ABB RAPID module: Module1.mod

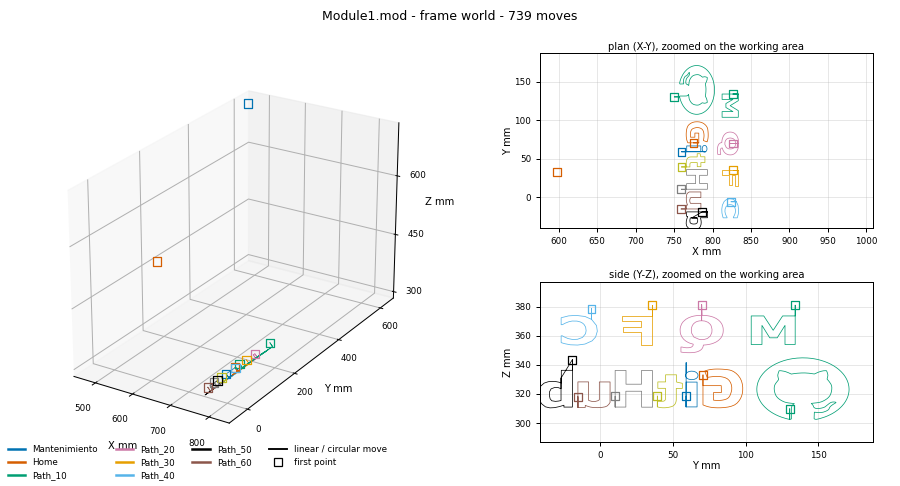
[picture p0: tool path of Module1.mod in frame world, 739 of 739 moves have a stored position in this frame; points joined in program order, loops and branches not executed]
MODULE Module1
    PERS tooldata TCP_Marcador:=[TRUE,[[70.711,0,142.836],[0.923879533,0,0.382683432,0]],[0.1,[0,0,1],[1,0,0,0],0,0,0]];
    PERS wobjdata Workobject_3:=[FALSE,TRUE,"",[[882.206,-55.622,379.617],[0.36650116,0,0.930417594,0]],[[0,0,0],[1,0,0,0]]];
    CONST robtarget Target_0:=[[81.772404685,689.476808944,-532.94398519],[0.776752007,-0.374117142,-0.504537271,-0.046204186],[0,0,-1,1],[9E+09,9E+09,9E+09,9E+09,9E+09,9E+09]];
    CONST robtarget Target_1:=[[84.162870332,88.825944226,-327.093570394],[0.96912891,0.008310335,0.246321364,-0.006773393],[0,-1,-1,0],[9E+09,9E+09,9E+09,9E+09,9E+09,9E+09]];
    CONST robtarget Target_50:=[[39.719,189.61,-28.8],[1,0,0,0],[-1,0,0,1],[9E+09,9E+09,9E+09,9E+09,9E+09,9E+09]];
    CONST robtarget Target_60:=[[39.719,180.982,-28.8],[1,0,0,0],[-1,0,0,1],[9E+09,9E+09,9E+09,9E+09,9E+09,9E+09]];
    CONST robtarget Target_70:=[[54.178,174.493,-28.8],[1,0,0,0],[-1,0,0,1],[9E+09,9E+09,9E+09,9E+09,9E+09,9E+09]];
    CONST robtarget Target_80:=[[39.719,168.028,-28.8],[1,0,0,0],[-1,0,0,1],[9E+09,9E+09,9E+09,9E+09,9E+09,9E+09]];
    CONST robtarget Target_180:=[[39.719,189.61,-38.8],[1,0,0,0],[-1,0,0,1],[9E+09,9E+09,9E+09,9E+09,9E+09,9E+09]];
    CONST robtarget Target_90:=[[39.719,159.4,-28.8],[1,0,0,0],[-1,0,0,1],[9E+09,9E+09,9E+09,9E+09,9E+09,9E+09]];
    CONST robtarget Target_100:=[[68.519,159.4,-28.8],[1,0,0,0],[-1,0,0,1],[9E+09,9E+09,9E+09,9E+09,9E+09,9E+09]];
    CONST robtarget Target_110:=[[68.519,166.782,-28.8],[1,0,0,0],[-1,0,0,1],[9E+09,9E+09,9E+09,9E+09,9E+09,9E+09]];
    CONST robtarget Target_120:=[[49.241,166.782,-28.8],[1,0,0,0],[-1,0,0,1],[9E+09,9E+09,9E+09,9E+09,9E+09,9E+09]];
    CONST robtarget Target_130:=[[61.748,172.119,-28.8],[1,0,0,0],[-1,0,0,1],[9E+09,9E+09,9E+09,9E+09,9E+09,9E+09]];
    CONST robtarget Target_140:=[[61.748,177.267,-28.8],[1,0,0,0],[-1,0,0,1],[9E+09,9E+09,9E+09,9E+09,9E+09,9E+09]];
    CONST robtarget Target_150:=[[49.241,182.604,-28.8],[1,0,0,0],[-1,0,0,1],[9E+09,9E+09,9E+09,9E+09,9E+09,9E+09]];
    CONST robtarget Target_160:=[[68.519,182.604,-28.8],[1,0,0,0],[-1,0,0,1],[9E+09,9E+09,9E+09,9E+09,9E+09,9E+09]];
    CONST robtarget Target_170:=[[68.519,189.61,-28.8],[1,0,0,0],[-1,0,0,1],[9E+09,9E+09,9E+09,9E+09,9E+09,9E+09]];
    CONST robtarget Target_970:=[[39.108,125.357,-38.8],[1,0,0,0],[-1,0,0,1],[9E+09,9E+09,9E+09,9E+09,9E+09,9E+09]];
    CONST robtarget Target_210:=[[39.108,125.357,-28.8],[1,0,0,0],[-1,0,0,1],[9E+09,9E+09,9E+09,9E+09,9E+09,9E+09]];
    CONST robtarget Target_220:=[[39.179,123.567,-28.8],[1,0,0,0],[-1,0,0,1],[9E+09,9E+09,9E+09,9E+09,9E+09,9E+09]];
    CONST robtarget Target_230:=[[39.408,121.803,-28.8],[1,0,0,0],[-1,0,0,1],[9E+09,9E+09,9E+09,9E+09,9E+09,9E+09]];
    CONST robtarget Target_240:=[[39.83,120.034,-28.8],[1,0,0,0],[-1,0,0,1],[9E+09,9E+09,9E+09,9E+09,9E+09,9E+09]];
    CONST robtarget Target_250:=[[40.454,118.354,-28.8],[1,0,0,0],[-1,0,0,1],[9E+09,9E+09,9E+09,9E+09,9E+09,9E+09]];
    CONST robtarget Target_260:=[[41.532,116.411,-28.8],[1,0,0,0],[-1,0,0,1],[9E+09,9E+09,9E+09,9E+09,9E+09,9E+09]];
    CONST robtarget Target_270:=[[43.092,114.53,-28.8],[1,0,0,0],[-1,0,0,1],[9E+09,9E+09,9E+09,9E+09,9E+09,9E+09]];
    CONST robtarget Target_280:=[[45.482,112.662,-28.8],[1,0,0,0],[-1,0,0,1],[9E+09,9E+09,9E+09,9E+09,9E+09,9E+09]];
    CONST robtarget Target_290:=[[47.725,111.578,-28.8],[1,0,0,0],[-1,0,0,1],[9E+09,9E+09,9E+09,9E+09,9E+09,9E+09]];
    CONST robtarget Target_300:=[[50.763,110.781,-28.8],[1,0,0,0],[-1,0,0,1],[9E+09,9E+09,9E+09,9E+09,9E+09,9E+09]];
    CONST robtarget Target_310:=[[53.109,110.544,-28.8],[1,0,0,0],[-1,0,0,1],[9E+09,9E+09,9E+09,9E+09,9E+09,9E+09]];
    CONST robtarget Target_320:=[[56.336,110.636,-28.8],[1,0,0,0],[-1,0,0,1],[9E+09,9E+09,9E+09,9E+09,9E+09,9E+09]];
    CONST robtarget Target_330:=[[58.625,111.031,-28.8],[1,0,0,0],[-1,0,0,1],[9E+09,9E+09,9E+09,9E+09,9E+09,9E+09]];
    CONST robtarget Target_340:=[[61.323,111.956,-28.8],[1,0,0,0],[-1,0,0,1],[9E+09,9E+09,9E+09,9E+09,9E+09,9E+09]];
    CONST robtarget Target_350:=[[63.282,113.038,-28.8],[1,0,0,0],[-1,0,0,1],[9E+09,9E+09,9E+09,9E+09,9E+09,9E+09]];
    CONST robtarget Target_360:=[[65.08,114.497,-28.8],[1,0,0,0],[-1,0,0,1],[9E+09,9E+09,9E+09,9E+09,9E+09,9E+09]];
    CONST robtarget Target_370:=[[66.459,116.132,-28.8],[1,0,0,0],[-1,0,0,1],[9E+09,9E+09,9E+09,9E+09,9E+09,9E+09]];
    CONST robtarget Target_380:=[[67.164,117.267,-28.8],[1,0,0,0],[-1,0,0,1],[9E+09,9E+09,9E+09,9E+09,9E+09,9E+09]];
    CONST robtarget Target_390:=[[68.166,119.573,-28.8],[1,0,0,0],[-1,0,0,1],[9E+09,9E+09,9E+09,9E+09,9E+09,9E+09]];
    CONST robtarget Target_400:=[[69.178,119.46,-28.8],[1,0,0,0],[-1,0,0,1],[9E+09,9E+09,9E+09,9E+09,9E+09,9E+09]];
    CONST robtarget Target_410:=[[70.001,119.208,-28.8],[1,0,0,0],[-1,0,0,1],[9E+09,9E+09,9E+09,9E+09,9E+09,9E+09]];
    CONST robtarget Target_420:=[[71.14,118.275,-28.8],[1,0,0,0],[-1,0,0,1],[9E+09,9E+09,9E+09,9E+09,9E+09,9E+09]];
    CONST robtarget Target_430:=[[71.611,117.079,-28.8],[1,0,0,0],[-1,0,0,1],[9E+09,9E+09,9E+09,9E+09,9E+09,9E+09]];
    CONST robtarget Target_440:=[[71.755,116.083,-28.8],[1,0,0,0],[-1,0,0,1],[9E+09,9E+09,9E+09,9E+09,9E+09,9E+09]];
    CONST robtarget Target_450:=[[71.779,114.935,-28.8],[1,0,0,0],[-1,0,0,1],[9E+09,9E+09,9E+09,9E+09,9E+09,9E+09]];
    CONST robtarget Target_460:=[[71.682,114.116,-28.8],[1,0,0,0],[-1,0,0,1],[9E+09,9E+09,9E+09,9E+09,9E+09,9E+09]];
    CONST robtarget Target_470:=[[71.431,113.012,-28.8],[1,0,0,0],[-1,0,0,1],[9E+09,9E+09,9E+09,9E+09,9E+09,9E+09]];
    CONST robtarget Target_480:=[[71.088,111.954,-28.8],[1,0,0,0],[-1,0,0,1],[9E+09,9E+09,9E+09,9E+09,9E+09,9E+09]];
    CONST robtarget Target_490:=[[71.034,111.11,-28.8],[1,0,0,0],[-1,0,0,1],[9E+09,9E+09,9E+09,9E+09,9E+09,9E+09]];
    CONST robtarget Target_500:=[[76.113,111.11,-28.8],[1,0,0,0],[-1,0,0,1],[9E+09,9E+09,9E+09,9E+09,9E+09,9E+09]];
    CONST robtarget Target_510:=[[76.379,112.375,-28.8],[1,0,0,0],[-1,0,0,1],[9E+09,9E+09,9E+09,9E+09,9E+09,9E+09]];
    CONST robtarget Target_520:=[[76.601,113.778,-28.8],[1,0,0,0],[-1,0,0,1],[9E+09,9E+09,9E+09,9E+09,9E+09,9E+09]];
    CONST robtarget Target_530:=[[76.712,115.33,-28.8],[1,0,0,0],[-1,0,0,1],[9E+09,9E+09,9E+09,9E+09,9E+09,9E+09]];
    CONST robtarget Target_540:=[[76.744,116.635,-28.8],[1,0,0,0],[-1,0,0,1],[9E+09,9E+09,9E+09,9E+09,9E+09,9E+09]];
    CONST robtarget Target_550:=[[76.732,118.083,-28.8],[1,0,0,0],[-1,0,0,1],[9E+09,9E+09,9E+09,9E+09,9E+09,9E+09]];
    CONST robtarget Target_560:=[[76.566,119.74,-28.8],[1,0,0,0],[-1,0,0,1],[9E+09,9E+09,9E+09,9E+09,9E+09,9E+09]];
    CONST robtarget Target_570:=[[76.396,120.574,-28.8],[1,0,0,0],[-1,0,0,1],[9E+09,9E+09,9E+09,9E+09,9E+09,9E+09]];
    CONST robtarget Target_580:=[[76.072,121.628,-28.8],[1,0,0,0],[-1,0,0,1],[9E+09,9E+09,9E+09,9E+09,9E+09,9E+09]];
    CONST robtarget Target_590:=[[75.527,122.831,-28.8],[1,0,0,0],[-1,0,0,1],[9E+09,9E+09,9E+09,9E+09,9E+09,9E+09]];
    CONST robtarget Target_600:=[[74.714,124.028,-28.8],[1,0,0,0],[-1,0,0,1],[9E+09,9E+09,9E+09,9E+09,9E+09,9E+09]];
    CONST robtarget Target_610:=[[73.676,125.003,-28.8],[1,0,0,0],[-1,0,0,1],[9E+09,9E+09,9E+09,9E+09,9E+09,9E+09]];
    CONST robtarget Target_620:=[[72.556,125.689,-28.8],[1,0,0,0],[-1,0,0,1],[9E+09,9E+09,9E+09,9E+09,9E+09,9E+09]];
    CONST robtarget Target_630:=[[71.041,126.234,-28.8],[1,0,0,0],[-1,0,0,1],[9E+09,9E+09,9E+09,9E+09,9E+09,9E+09]];
    CONST robtarget Target_640:=[[69.456,126.502,-28.8],[1,0,0,0],[-1,0,0,1],[9E+09,9E+09,9E+09,9E+09,9E+09,9E+09]];
    CONST robtarget Target_650:=[[69.036,126.532,-28.8],[1,0,0,0],[-1,0,0,1],[9E+09,9E+09,9E+09,9E+09,9E+09,9E+09]];
    CONST robtarget Target_660:=[[68.932,127.738,-28.8],[1,0,0,0],[-1,0,0,1],[9E+09,9E+09,9E+09,9E+09,9E+09,9E+09]];
    CONST robtarget Target_670:=[[68.743,128.995,-28.8],[1,0,0,0],[-1,0,0,1],[9E+09,9E+09,9E+09,9E+09,9E+09,9E+09]];
    CONST robtarget Target_680:=[[68.43,130.365,-28.8],[1,0,0,0],[-1,0,0,1],[9E+09,9E+09,9E+09,9E+09,9E+09,9E+09]];
    CONST robtarget Target_690:=[[67.943,131.835,-28.8],[1,0,0,0],[-1,0,0,1],[9E+09,9E+09,9E+09,9E+09,9E+09,9E+09]];
    CONST robtarget Target_700:=[[67.321,133.199,-28.8],[1,0,0,0],[-1,0,0,1],[9E+09,9E+09,9E+09,9E+09,9E+09,9E+09]];
    CONST robtarget Target_710:=[[66.175,134.99,-28.8],[1,0,0,0],[-1,0,0,1],[9E+09,9E+09,9E+09,9E+09,9E+09,9E+09]];
    CONST robtarget Target_720:=[[65.544,135.746,-28.8],[1,0,0,0],[-1,0,0,1],[9E+09,9E+09,9E+09,9E+09,9E+09,9E+09]];
    CONST robtarget Target_730:=[[64.638,136.648,-28.8],[1,0,0,0],[-1,0,0,1],[9E+09,9E+09,9E+09,9E+09,9E+09,9E+09]];
    CONST robtarget Target_740:=[[64.061,137.137,-28.8],[1,0,0,0],[-1,0,0,1],[9E+09,9E+09,9E+09,9E+09,9E+09,9E+09]];
    CONST robtarget Target_750:=[[62.566,138.163,-28.8],[1,0,0,0],[-1,0,0,1],[9E+09,9E+09,9E+09,9E+09,9E+09,9E+09]];
    CONST robtarget Target_760:=[[61.546,138.701,-28.8],[1,0,0,0],[-1,0,0,1],[9E+09,9E+09,9E+09,9E+09,9E+09,9E+09]];
    CONST robtarget Target_770:=[[60.255,139.232,-28.8],[1,0,0,0],[-1,0,0,1],[9E+09,9E+09,9E+09,9E+09,9E+09,9E+09]];
    CONST robtarget Target_780:=[[59.077,139.596,-28.8],[1,0,0,0],[-1,0,0,1],[9E+09,9E+09,9E+09,9E+09,9E+09,9E+09]];
    CONST robtarget Target_790:=[[57.514,139.929,-28.8],[1,0,0,0],[-1,0,0,1],[9E+09,9E+09,9E+09,9E+09,9E+09,9E+09]];
    CONST robtarget Target_800:=[[56.02,140.114,-28.8],[1,0,0,0],[-1,0,0,1],[9E+09,9E+09,9E+09,9E+09,9E+09,9E+09]];
    CONST robtarget Target_810:=[[54.254,140.191,-28.8],[1,0,0,0],[-1,0,0,1],[9E+09,9E+09,9E+09,9E+09,9E+09,9E+09]];
    CONST robtarget Target_820:=[[52.801,140.154,-28.8],[1,0,0,0],[-1,0,0,1],[9E+09,9E+09,9E+09,9E+09,9E+09,9E+09]];
    CONST robtarget Target_830:=[[51.332,140.017,-28.8],[1,0,0,0],[-1,0,0,1],[9E+09,9E+09,9E+09,9E+09,9E+09,9E+09]];
    CONST robtarget Target_840:=[[49.345,139.643,-28.8],[1,0,0,0],[-1,0,0,1],[9E+09,9E+09,9E+09,9E+09,9E+09,9E+09]];
    CONST robtarget Target_850:=[[47.546,139.074,-28.8],[1,0,0,0],[-1,0,0,1],[9E+09,9E+09,9E+09,9E+09,9E+09,9E+09]];
    CONST robtarget Target_860:=[[45.602,138.136,-28.8],[1,0,0,0],[-1,0,0,1],[9E+09,9E+09,9E+09,9E+09,9E+09,9E+09]];
    CONST robtarget Target_870:=[[43.821,136.874,-28.8],[1,0,0,0],[-1,0,0,1],[9E+09,9E+09,9E+09,9E+09,9E+09,9E+09]];
    CONST robtarget Target_880:=[[42.287,135.334,-28.8],[1,0,0,0],[-1,0,0,1],[9E+09,9E+09,9E+09,9E+09,9E+09,9E+09]];
    CONST robtarget Target_890:=[[41.065,133.588,-28.8],[1,0,0,0],[-1,0,0,1],[9E+09,9E+09,9E+09,9E+09,9E+09,9E+09]];
    CONST robtarget Target_900:=[[40.433,132.344,-28.8],[1,0,0,0],[-1,0,0,1],[9E+09,9E+09,9E+09,9E+09,9E+09,9E+09]];
    CONST robtarget Target_910:=[[39.916,130.983,-28.8],[1,0,0,0],[-1,0,0,1],[9E+09,9E+09,9E+09,9E+09,9E+09,9E+09]];
    CONST robtarget Target_920:=[[39.561,129.683,-28.8],[1,0,0,0],[-1,0,0,1],[9E+09,9E+09,9E+09,9E+09,9E+09,9E+09]];
    CONST robtarget Target_930:=[[39.367,128.69,-28.8],[1,0,0,0],[-1,0,0,1],[9E+09,9E+09,9E+09,9E+09,9E+09,9E+09]];
    CONST robtarget Target_940:=[[39.19,127.284,-28.8],[1,0,0,0],[-1,0,0,1],[9E+09,9E+09,9E+09,9E+09,9E+09,9E+09]];
    CONST robtarget Target_950:=[[39.132,126.428,-28.8],[1,0,0,0],[-1,0,0,1],[9E+09,9E+09,9E+09,9E+09,9E+09,9E+09]];
    CONST robtarget Target_960:=[[39.109,125.612,-28.8],[1,0,0,0],[-1,0,0,1],[9E+09,9E+09,9E+09,9E+09,9E+09,9E+09]];
    CONST robtarget Target_1360:=[[44.538,125.357,-38.8],[1,0,0,0],[-1,0,0,1],[9E+09,9E+09,9E+09,9E+09,9E+09,9E+09]];
    CONST robtarget Target_1370:=[[44.538,125.357,-28.8],[1,0,0,0],[-1,0,0,1],[9E+09,9E+09,9E+09,9E+09,9E+09,9E+09]];
    CONST robtarget Target_1380:=[[44.718,123.741,-28.8],[1,0,0,0],[-1,0,0,1],[9E+09,9E+09,9E+09,9E+09,9E+09,9E+09]];
    CONST robtarget Target_1390:=[[45.229,122.281,-28.8],[1,0,0,0],[-1,0,0,1],[9E+09,9E+09,9E+09,9E+09,9E+09,9E+09]];
    CONST robtarget Target_1400:=[[46.016,121.112,-28.8],[1,0,0,0],[-1,0,0,1],[9E+09,9E+09,9E+09,9E+09,9E+09,9E+09]];
    CONST robtarget Target_1410:=[[47.526,119.826,-28.8],[1,0,0,0],[-1,0,0,1],[9E+09,9E+09,9E+09,9E+09,9E+09,9E+09]];
    CONST robtarget Target_1420:=[[49.143,119.027,-28.8],[1,0,0,0],[-1,0,0,1],[9E+09,9E+09,9E+09,9E+09,9E+09,9E+09]];
    CONST robtarget Target_1430:=[[51.333,118.437,-28.8],[1,0,0,0],[-1,0,0,1],[9E+09,9E+09,9E+09,9E+09,9E+09,9E+09]];
    CONST robtarget Target_1440:=[[53.838,118.235,-28.8],[1,0,0,0],[-1,0,0,1],[9E+09,9E+09,9E+09,9E+09,9E+09,9E+09]];
    CONST robtarget Target_1450:=[[57.053,118.466,-28.8],[1,0,0,0],[-1,0,0,1],[9E+09,9E+09,9E+09,9E+09,9E+09,9E+09]];
    CONST robtarget Target_1460:=[[60.981,120.015,-28.8],[1,0,0,0],[-1,0,0,1],[9E+09,9E+09,9E+09,9E+09,9E+09,9E+09]];
    CONST robtarget Target_1470:=[[63.547,124.003,-28.8],[1,0,0,0],[-1,0,0,1],[9E+09,9E+09,9E+09,9E+09,9E+09,9E+09]];
    CONST robtarget Target_1480:=[[63.533,126.78,-28.8],[1,0,0,0],[-1,0,0,1],[9E+09,9E+09,9E+09,9E+09,9E+09,9E+09]];
    CONST robtarget Target_1490:=[[62.461,129.265,-28.8],[1,0,0,0],[-1,0,0,1],[9E+09,9E+09,9E+09,9E+09,9E+09,9E+09]];
    CONST robtarget Target_1500:=[[59.965,131.302,-28.8],[1,0,0,0],[-1,0,0,1],[9E+09,9E+09,9E+09,9E+09,9E+09,9E+09]];
    CONST robtarget Target_1510:=[[56.224,132.368,-28.8],[1,0,0,0],[-1,0,0,1],[9E+09,9E+09,9E+09,9E+09,9E+09,9E+09]];
    CONST robtarget Target_1520:=[[53.223,132.461,-28.8],[1,0,0,0],[-1,0,0,1],[9E+09,9E+09,9E+09,9E+09,9E+09,9E+09]];
    CONST robtarget Target_1530:=[[49.744,131.887,-28.8],[1,0,0,0],[-1,0,0,1],[9E+09,9E+09,9E+09,9E+09,9E+09,9E+09]];
    CONST robtarget Target_1580:=[[48.111,131.233,-28.8],[1,0,0,0],[-1,0,0,1],[9E+09,9E+09,9E+09,9E+09,9E+09,9E+09]];
    CONST robtarget Target_1590:=[[46.155,129.752,-28.8],[1,0,0,0],[-1,0,0,1],[9E+09,9E+09,9E+09,9E+09,9E+09,9E+09]];
    CONST robtarget Target_1600:=[[44.889,127.593,-28.8],[1,0,0,0],[-1,0,0,1],[9E+09,9E+09,9E+09,9E+09,9E+09,9E+09]];
    CONST robtarget Target_1610:=[[39.719,91.314,-38.8],[1,0,0,0],[-1,0,0,1],[9E+09,9E+09,9E+09,9E+09,9E+09,9E+09]];
    CONST robtarget Target_1620:=[[39.719,91.314,-28.8],[1,0,0,0],[-1,0,0,1],[9E+09,9E+09,9E+09,9E+09,9E+09,9E+09]];
    CONST robtarget Target_1630:=[[39.719,70.672,-28.8],[1,0,0,0],[-1,0,0,1],[9E+09,9E+09,9E+09,9E+09,9E+09,9E+09]];
    CONST robtarget Target_1640:=[[45.291,70.672,-28.8],[1,0,0,0],[-1,0,0,1],[9E+09,9E+09,9E+09,9E+09,9E+09,9E+09]];
    CONST robtarget Target_1650:=[[45.291,83.932,-28.8],[1,0,0,0],[-1,0,0,1],[9E+09,9E+09,9E+09,9E+09,9E+09,9E+09]];
    CONST robtarget Target_1660:=[[50.651,83.932,-28.8],[1,0,0,0],[-1,0,0,1],[9E+09,9E+09,9E+09,9E+09,9E+09,9E+09]];
    CONST robtarget Target_1670:=[[50.651,71.636,-28.8],[1,0,0,0],[-1,0,0,1],[9E+09,9E+09,9E+09,9E+09,9E+09,9E+09]];
    CONST robtarget Target_1680:=[[56.223,71.636,-28.8],[1,0,0,0],[-1,0,0,1],[9E+09,9E+09,9E+09,9E+09,9E+09,9E+09]];
    CONST robtarget Target_1690:=[[56.223,83.932,-28.8],[1,0,0,0],[-1,0,0,1],[9E+09,9E+09,9E+09,9E+09,9E+09,9E+09]];
    CONST robtarget Target_1700:=[[68.519,83.932,-28.8],[1,0,0,0],[-1,0,0,1],[9E+09,9E+09,9E+09,9E+09,9E+09,9E+09]];
    CONST robtarget Target_1710:=[[68.519,91.314,-28.8],[1,0,0,0],[-1,0,0,1],[9E+09,9E+09,9E+09,9E+09,9E+09,9E+09]];
    CONST robtarget Target_1720:=[[43.151,49.677,-38.8],[1,0,0,0],[-1,0,0,1],[9E+09,9E+09,9E+09,9E+09,9E+09,9E+09]];
    CONST robtarget Target_1730:=[[43.151,49.677,-28.8],[1,0,0,0],[-1,0,0,1],[9E+09,9E+09,9E+09,9E+09,9E+09,9E+09]];
    CONST robtarget Target_1740:=[[40.268,45.197,-28.8],[1,0,0,0],[-1,0,0,1],[9E+09,9E+09,9E+09,9E+09,9E+09,9E+09]];
    CONST robtarget Target_1750:=[[39.155,39.012,-28.8],[1,0,0,0],[-1,0,0,1],[9E+09,9E+09,9E+09,9E+09,9E+09,9E+09]];
    CONST robtarget Target_1760:=[[39.66,33.924,-28.8],[1,0,0,0],[-1,0,0,1],[9E+09,9E+09,9E+09,9E+09,9E+09,9E+09]];
    CONST robtarget Target_1770:=[[41.553,28.8,-28.8],[1,0,0,0],[-1,0,0,1],[9E+09,9E+09,9E+09,9E+09,9E+09,9E+09]];
    CONST robtarget Target_1780:=[[48.535,28.8,-28.8],[1,0,0,0],[-1,0,0,1],[9E+09,9E+09,9E+09,9E+09,9E+09,9E+09]];
    CONST robtarget Target_1790:=[[48.535,29.647,-28.8],[1,0,0,0],[-1,0,0,1],[9E+09,9E+09,9E+09,9E+09,9E+09,9E+09]];
    CONST robtarget Target_1800:=[[46.954,31.662,-28.8],[1,0,0,0],[-1,0,0,1],[9E+09,9E+09,9E+09,9E+09,9E+09,9E+09]];
    CONST robtarget Target_1810:=[[45.633,33.957,-28.8],[1,0,0,0],[-1,0,0,1],[9E+09,9E+09,9E+09,9E+09,9E+09,9E+09]];
    CONST robtarget Target_1820:=[[44.85,36.357,-28.8],[1,0,0,0],[-1,0,0,1],[9E+09,9E+09,9E+09,9E+09,9E+09,9E+09]];
    CONST robtarget Target_1830:=[[44.913,39.686,-28.8],[1,0,0,0],[-1,0,0,1],[9E+09,9E+09,9E+09,9E+09,9E+09,9E+09]];
    CONST robtarget Target_1840:=[[45.786,42.02,-28.8],[1,0,0,0],[-1,0,0,1],[9E+09,9E+09,9E+09,9E+09,9E+09,9E+09]];
    CONST robtarget Target_1850:=[[47.007,43.565,-28.8],[1,0,0,0],[-1,0,0,1],[9E+09,9E+09,9E+09,9E+09,9E+09,9E+09]];
    CONST robtarget Target_1860:=[[48.266,44.527,-28.8],[1,0,0,0],[-1,0,0,1],[9E+09,9E+09,9E+09,9E+09,9E+09,9E+09]];
    CONST robtarget Target_1870:=[[50.968,45.626,-28.8],[1,0,0,0],[-1,0,0,1],[9E+09,9E+09,9E+09,9E+09,9E+09,9E+09]];
    CONST robtarget Target_1880:=[[54.572,45.959,-28.8],[1,0,0,0],[-1,0,0,1],[9E+09,9E+09,9E+09,9E+09,9E+09,9E+09]];
    CONST robtarget Target_1890:=[[57.659,45.553,-28.8],[1,0,0,0],[-1,0,0,1],[9E+09,9E+09,9E+09,9E+09,9E+09,9E+09]];
    CONST robtarget Target_1900:=[[61.355,43.476,-28.8],[1,0,0,0],[-1,0,0,1],[9E+09,9E+09,9E+09,9E+09,9E+09,9E+09]];
    CONST robtarget Target_1910:=[[63.218,40.068,-28.8],[1,0,0,0],[-1,0,0,1],[9E+09,9E+09,9E+09,9E+09,9E+09,9E+09]];
    CONST robtarget Target_1920:=[[63.451,36.743,-28.8],[1,0,0,0],[-1,0,0,1],[9E+09,9E+09,9E+09,9E+09,9E+09,9E+09]];
    CONST robtarget Target_1930:=[[62.507,33.56,-28.8],[1,0,0,0],[-1,0,0,1],[9E+09,9E+09,9E+09,9E+09,9E+09,9E+09]];
    CONST robtarget Target_1940:=[[60.82,30.89,-28.8],[1,0,0,0],[-1,0,0,1],[9E+09,9E+09,9E+09,9E+09,9E+09,9E+09]];
    CONST robtarget Target_1950:=[[59.726,29.576,-28.8],[1,0,0,0],[-1,0,0,1],[9E+09,9E+09,9E+09,9E+09,9E+09,9E+09]];
    CONST robtarget Target_1960:=[[59.726,28.8,-28.8],[1,0,0,0],[-1,0,0,1],[9E+09,9E+09,9E+09,9E+09,9E+09,9E+09]];
    CONST robtarget Target_1970:=[[66.615,28.8,-28.8],[1,0,0,0],[-1,0,0,1],[9E+09,9E+09,9E+09,9E+09,9E+09,9E+09]];
    CONST robtarget Target_1980:=[[67.669,31.258,-28.8],[1,0,0,0],[-1,0,0,1],[9E+09,9E+09,9E+09,9E+09,9E+09,9E+09]];
    CONST robtarget Target_1990:=[[68.783,35.103,-28.8],[1,0,0,0],[-1,0,0,1],[9E+09,9E+09,9E+09,9E+09,9E+09,9E+09]];
    CONST robtarget Target_2000:=[[69.052,40.129,-28.8],[1,0,0,0],[-1,0,0,1],[9E+09,9E+09,9E+09,9E+09,9E+09,9E+09]];
    CONST robtarget Target_2010:=[[68.022,45.218,-28.8],[1,0,0,0],[-1,0,0,1],[9E+09,9E+09,9E+09,9E+09,9E+09,9E+09]];
    CONST robtarget Target_2020:=[[64.819,50.073,-28.8],[1,0,0,0],[-1,0,0,1],[9E+09,9E+09,9E+09,9E+09,9E+09,9E+09]];
    CONST robtarget Target_2030:=[[60.925,52.489,-28.8],[1,0,0,0],[-1,0,0,1],[9E+09,9E+09,9E+09,9E+09,9E+09,9E+09]];
    CONST robtarget Target_2040:=[[55.153,53.654,-28.8],[1,0,0,0],[-1,0,0,1],[9E+09,9E+09,9E+09,9E+09,9E+09,9E+09]];
    CONST robtarget Target_2050:=[[49.431,53.115,-28.8],[1,0,0,0],[-1,0,0,1],[9E+09,9E+09,9E+09,9E+09,9E+09,9E+09]];
    CONST robtarget Target_2060:=[[94.492,36.518,-38.8],[1,0,0,0],[-1,0,0,1],[9E+09,9E+09,9E+09,9E+09,9E+09,9E+09]];
    CONST robtarget Target_2070:=[[94.492,36.518,-28.8],[1,0,0,0],[-1,0,0,1],[9E+09,9E+09,9E+09,9E+09,9E+09,9E+09]];
    CONST robtarget Target_2080:=[[94.492,28.907,-28.8],[1,0,0,0],[-1,0,0,1],[9E+09,9E+09,9E+09,9E+09,9E+09,9E+09]];
    CONST robtarget Target_2090:=[[107.157,28.907,-28.8],[1,0,0,0],[-1,0,0,1],[9E+09,9E+09,9E+09,9E+09,9E+09,9E+09]];
    CONST robtarget Target_2100:=[[106.387,27.012,-28.8],[1,0,0,0],[-1,0,0,1],[9E+09,9E+09,9E+09,9E+09,9E+09,9E+09]];
    CONST robtarget Target_2110:=[[105.808,24.978,-28.8],[1,0,0,0],[-1,0,0,1],[9E+09,9E+09,9E+09,9E+09,9E+09,9E+09]];
    CONST robtarget Target_2120:=[[105.615,22.663,-28.8],[1,0,0,0],[-1,0,0,1],[9E+09,9E+09,9E+09,9E+09,9E+09,9E+09]];
    CONST robtarget Target_2130:=[[105.998,19.953,-28.8],[1,0,0,0],[-1,0,0,1],[9E+09,9E+09,9E+09,9E+09,9E+09,9E+09]];
    CONST robtarget Target_2140:=[[107.388,17.105,-28.8],[1,0,0,0],[-1,0,0,1],[9E+09,9E+09,9E+09,9E+09,9E+09,9E+09]];
    CONST robtarget Target_2150:=[[110.564,14.681,-28.8],[1,0,0,0],[-1,0,0,1],[9E+09,9E+09,9E+09,9E+09,9E+09,9E+09]];
    CONST robtarget Target_2160:=[[116.326,13.247,-28.8],[1,0,0,0],[-1,0,0,1],[9E+09,9E+09,9E+09,9E+09,9E+09,9E+09]];
    CONST robtarget Target_2170:=[[122.982,13.464,-28.8],[1,0,0,0],[-1,0,0,1],[9E+09,9E+09,9E+09,9E+09,9E+09,9E+09]];
    CONST robtarget Target_2180:=[[128.107,15.275,-28.8],[1,0,0,0],[-1,0,0,1],[9E+09,9E+09,9E+09,9E+09,9E+09,9E+09]];
    CONST robtarget Target_2190:=[[131.293,18.015,-28.8],[1,0,0,0],[-1,0,0,1],[9E+09,9E+09,9E+09,9E+09,9E+09,9E+09]];
    CONST robtarget Target_2200:=[[132.343,21.11,-28.8],[1,0,0,0],[-1,0,0,1],[9E+09,9E+09,9E+09,9E+09,9E+09,9E+09]];
    CONST robtarget Target_2210:=[[132.102,24.275,-28.8],[1,0,0,0],[-1,0,0,1],[9E+09,9E+09,9E+09,9E+09,9E+09,9E+09]];
    CONST robtarget Target_2220:=[[131.088,27.483,-28.8],[1,0,0,0],[-1,0,0,1],[9E+09,9E+09,9E+09,9E+09,9E+09,9E+09]];
    CONST robtarget Target_2230:=[[129.679,30.716,-28.8],[1,0,0,0],[-1,0,0,1],[9E+09,9E+09,9E+09,9E+09,9E+09,9E+09]];
    CONST robtarget Target_2240:=[[131.55,30.716,-28.8],[1,0,0,0],[-1,0,0,1],[9E+09,9E+09,9E+09,9E+09,9E+09,9E+09]];
    CONST robtarget Target_2250:=[[131.55,36.518,-28.8],[1,0,0,0],[-1,0,0,1],[9E+09,9E+09,9E+09,9E+09,9E+09,9E+09]];
    CONST robtarget Target_2260:=[[113.021,28.72,-38.8],[1,0,0,0],[-1,0,0,1],[9E+09,9E+09,9E+09,9E+09,9E+09,9E+09]];
    CONST robtarget Target_2270:=[[113.021,28.72,-28.8],[1,0,0,0],[-1,0,0,1],[9E+09,9E+09,9E+09,9E+09,9E+09,9E+09]];
    CONST robtarget Target_2280:=[[111.875,26.718,-28.8],[1,0,0,0],[-1,0,0,1],[9E+09,9E+09,9E+09,9E+09,9E+09,9E+09]];
    CONST robtarget Target_2290:=[[111.898,24.166,-28.8],[1,0,0,0],[-1,0,0,1],[9E+09,9E+09,9E+09,9E+09,9E+09,9E+09]];
    CONST robtarget Target_2300:=[[113.178,21.908,-28.8],[1,0,0,0],[-1,0,0,1],[9E+09,9E+09,9E+09,9E+09,9E+09,9E+09]];
    CONST robtarget Target_2310:=[[116.016,20.859,-28.8],[1,0,0,0],[-1,0,0,1],[9E+09,9E+09,9E+09,9E+09,9E+09,9E+09]];
    CONST robtarget Target_2320:=[[120.005,20.743,-28.8],[1,0,0,0],[-1,0,0,1],[9E+09,9E+09,9E+09,9E+09,9E+09,9E+09]];
    CONST robtarget Target_2330:=[[123.183,21.23,-28.8],[1,0,0,0],[-1,0,0,1],[9E+09,9E+09,9E+09,9E+09,9E+09,9E+09]];
    CONST robtarget Target_2340:=[[125.187,22.357,-28.8],[1,0,0,0],[-1,0,0,1],[9E+09,9E+09,9E+09,9E+09,9E+09,9E+09]];
    CONST robtarget Target_2350:=[[125.791,24.868,-28.8],[1,0,0,0],[-1,0,0,1],[9E+09,9E+09,9E+09,9E+09,9E+09,9E+09]];
    CONST robtarget Target_2360:=[[125.52,26.754,-28.8],[1,0,0,0],[-1,0,0,1],[9E+09,9E+09,9E+09,9E+09,9E+09,9E+09]];
    CONST robtarget Target_2370:=[[124.999,28.72,-28.8],[1,0,0,0],[-1,0,0,1],[9E+09,9E+09,9E+09,9E+09,9E+09,9E+09]];
    CONST robtarget Target_2380:=[[131.862,40.324,-38.8],[1,0,0,0],[-1,0,0,1],[9E+09,9E+09,9E+09,9E+09,9E+09,9E+09]];
    CONST robtarget Target_2390:=[[131.862,40.324,-28.8],[1,0,0,0],[-1,0,0,1],[9E+09,9E+09,9E+09,9E+09,9E+09,9E+09]];
    CONST robtarget Target_2400:=[[106.159,40.324,-28.8],[1,0,0,0],[-1,0,0,1],[9E+09,9E+09,9E+09,9E+09,9E+09,9E+09]];
    CONST robtarget Target_2410:=[[106.159,47.623,-28.8],[1,0,0,0],[-1,0,0,1],[9E+09,9E+09,9E+09,9E+09,9E+09,9E+09]];
    CONST robtarget Target_2420:=[[124.75,47.623,-28.8],[1,0,0,0],[-1,0,0,1],[9E+09,9E+09,9E+09,9E+09,9E+09,9E+09]];
    CONST robtarget Target_2430:=[[125.344,48.766,-28.8],[1,0,0,0],[-1,0,0,1],[9E+09,9E+09,9E+09,9E+09,9E+09,9E+09]];
    CONST robtarget Target_2440:=[[125.811,49.951,-28.8],[1,0,0,0],[-1,0,0,1],[9E+09,9E+09,9E+09,9E+09,9E+09,9E+09]];
    CONST robtarget Target_2450:=[[125.998,51.897,-28.8],[1,0,0,0],[-1,0,0,1],[9E+09,9E+09,9E+09,9E+09,9E+09,9E+09]];
    CONST robtarget Target_2460:=[[125.169,53.997,-28.8],[1,0,0,0],[-1,0,0,1],[9E+09,9E+09,9E+09,9E+09,9E+09,9E+09]];
    CONST robtarget Target_2470:=[[124.156,55.047,-28.8],[1,0,0,0],[-1,0,0,1],[9E+09,9E+09,9E+09,9E+09,9E+09,9E+09]];
    CONST robtarget Target_2480:=[[106.221,55.047,-28.8],[1,0,0,0],[-1,0,0,1],[9E+09,9E+09,9E+09,9E+09,9E+09,9E+09]];
    CONST robtarget Target_2490:=[[106.221,62.409,-28.8],[1,0,0,0],[-1,0,0,1],[9E+09,9E+09,9E+09,9E+09,9E+09,9E+09]];
    CONST robtarget Target_2500:=[[126.871,62.409,-28.8],[1,0,0,0],[-1,0,0,1],[9E+09,9E+09,9E+09,9E+09,9E+09,9E+09]];
    CONST robtarget Target_2510:=[[128.785,61.552,-28.8],[1,0,0,0],[-1,0,0,1],[9E+09,9E+09,9E+09,9E+09,9E+09,9E+09]];
    CONST robtarget Target_2520:=[[130.427,60.381,-28.8],[1,0,0,0],[-1,0,0,1],[9E+09,9E+09,9E+09,9E+09,9E+09,9E+09]];
    CONST robtarget Target_2530:=[[131.301,58.995,-28.8],[1,0,0,0],[-1,0,0,1],[9E+09,9E+09,9E+09,9E+09,9E+09,9E+09]];
    CONST robtarget Target_2540:=[[131.874,56.704,-28.8],[1,0,0,0],[-1,0,0,1],[9E+09,9E+09,9E+09,9E+09,9E+09,9E+09]];
    CONST robtarget Target_2550:=[[132.12,53.899,-28.8],[1,0,0,0],[-1,0,0,1],[9E+09,9E+09,9E+09,9E+09,9E+09,9E+09]];
    CONST robtarget Target_2560:=[[132.002,51.051,-28.8],[1,0,0,0],[-1,0,0,1],[9E+09,9E+09,9E+09,9E+09,9E+09,9E+09]];
    CONST robtarget Target_2570:=[[131.494,48.781,-28.8],[1,0,0,0],[-1,0,0,1],[9E+09,9E+09,9E+09,9E+09,9E+09,9E+09]];
    CONST robtarget Target_2580:=[[130.719,46.967,-28.8],[1,0,0,0],[-1,0,0,1],[9E+09,9E+09,9E+09,9E+09,9E+09,9E+09]];
    CONST robtarget Target_2590:=[[129.803,45.377,-28.8],[1,0,0,0],[-1,0,0,1],[9E+09,9E+09,9E+09,9E+09,9E+09,9E+09]];
    CONST robtarget Target_2600:=[[131.862,45.377,-28.8],[1,0,0,0],[-1,0,0,1],[9E+09,9E+09,9E+09,9E+09,9E+09,9E+09]];
    CONST robtarget Target_2610:=[[131.528,65.918,-38.8],[1,0,0,0],[-1,0,0,1],[9E+09,9E+09,9E+09,9E+09,9E+09,9E+09]];
    CONST robtarget Target_2620:=[[131.528,65.918,-28.8],[1,0,0,0],[-1,0,0,1],[9E+09,9E+09,9E+09,9E+09,9E+09,9E+09]];
    CONST robtarget Target_2630:=[[94.623,65.918,-28.8],[1,0,0,0],[-1,0,0,1],[9E+09,9E+09,9E+09,9E+09,9E+09,9E+09]];
    CONST robtarget Target_2640:=[[94.623,73.366,-28.8],[1,0,0,0],[-1,0,0,1],[9E+09,9E+09,9E+09,9E+09,9E+09,9E+09]];
    CONST robtarget Target_2650:=[[108.5,73.366,-28.8],[1,0,0,0],[-1,0,0,1],[9E+09,9E+09,9E+09,9E+09,9E+09,9E+09]];
    CONST robtarget Target_2660:=[[108.5,84.029,-28.8],[1,0,0,0],[-1,0,0,1],[9E+09,9E+09,9E+09,9E+09,9E+09,9E+09]];
    CONST robtarget Target_2670:=[[94.623,84.029,-28.8],[1,0,0,0],[-1,0,0,1],[9E+09,9E+09,9E+09,9E+09,9E+09,9E+09]];
    CONST robtarget Target_2680:=[[94.623,91.485,-28.8],[1,0,0,0],[-1,0,0,1],[9E+09,9E+09,9E+09,9E+09,9E+09,9E+09]];
    CONST robtarget Target_2690:=[[131.64,91.652,-28.8],[1,0,0,0],[-1,0,0,1],[9E+09,9E+09,9E+09,9E+09,9E+09,9E+09]];
    CONST robtarget Target_2700:=[[131.64,84.093,-28.8],[1,0,0,0],[-1,0,0,1],[9E+09,9E+09,9E+09,9E+09,9E+09,9E+09]];
    CONST robtarget Target_2710:=[[115.577,84.093,-28.8],[1,0,0,0],[-1,0,0,1],[9E+09,9E+09,9E+09,9E+09,9E+09,9E+09]];
    CONST robtarget Target_2720:=[[115.577,73.257,-28.8],[1,0,0,0],[-1,0,0,1],[9E+09,9E+09,9E+09,9E+09,9E+09,9E+09]];
    CONST robtarget Target_2730:=[[131.528,73.257,-28.8],[1,0,0,0],[-1,0,0,1],[9E+09,9E+09,9E+09,9E+09,9E+09,9E+09]];
    CONST robtarget Target_2739:=[[131.262,94.901,-38.8],[1,0,0,0],[-1,0,0,1],[9E+09,9E+09,9E+09,9E+09,9E+09,9E+09]];
    CONST robtarget Target_2740:=[[131.262,94.901,-28.8],[1,0,0,0],[-1,0,0,1],[9E+09,9E+09,9E+09,9E+09,9E+09,9E+09]];
    CONST robtarget Target_2750:=[[131.469,95.335,-28.8],[1,0,0,0],[-1,0,0,1],[9E+09,9E+09,9E+09,9E+09,9E+09,9E+09]];
    CONST robtarget Target_2760:=[[131.67,95.797,-28.8],[1,0,0,0],[-1,0,0,1],[9E+09,9E+09,9E+09,9E+09,9E+09,9E+09]];
    CONST robtarget Target_2770:=[[131.853,96.314,-28.8],[1,0,0,0],[-1,0,0,1],[9E+09,9E+09,9E+09,9E+09,9E+09,9E+09]];
    CONST robtarget Target_2780:=[[132.01,96.915,-28.8],[1,0,0,0],[-1,0,0,1],[9E+09,9E+09,9E+09,9E+09,9E+09,9E+09]];
    CONST robtarget Target_2790:=[[132.134,97.627,-28.8],[1,0,0,0],[-1,0,0,1],[9E+09,9E+09,9E+09,9E+09,9E+09,9E+09]];
    CONST robtarget Target_2800:=[[132.214,98.479,-28.8],[1,0,0,0],[-1,0,0,1],[9E+09,9E+09,9E+09,9E+09,9E+09,9E+09]];
    CONST robtarget Target_2810:=[[132.242,99.498,-28.8],[1,0,0,0],[-1,0,0,1],[9E+09,9E+09,9E+09,9E+09,9E+09,9E+09]];
    CONST robtarget Target_2820:=[[132.178,100.608,-28.8],[1,0,0,0],[-1,0,0,1],[9E+09,9E+09,9E+09,9E+09,9E+09,9E+09]];
    CONST robtarget Target_2830:=[[132.01,101.688,-28.8],[1,0,0,0],[-1,0,0,1],[9E+09,9E+09,9E+09,9E+09,9E+09,9E+09]];
    CONST robtarget Target_2840:=[[131.761,102.707,-28.8],[1,0,0,0],[-1,0,0,1],[9E+09,9E+09,9E+09,9E+09,9E+09,9E+09]];
    CONST robtarget Target_2850:=[[131.469,103.613,-28.8],[1,0,0,0],[-1,0,0,1],[9E+09,9E+09,9E+09,9E+09,9E+09,9E+09]];
    CONST robtarget Target_2860:=[[131.169,104.387,-28.8],[1,0,0,0],[-1,0,0,1],[9E+09,9E+09,9E+09,9E+09,9E+09,9E+09]];
    CONST robtarget Target_2870:=[[130.893,104.981,-28.8],[1,0,0,0],[-1,0,0,1],[9E+09,9E+09,9E+09,9E+09,9E+09,9E+09]];
    CONST robtarget Target_2880:=[[130.668,105.355,-28.8],[1,0,0,0],[-1,0,0,1],[9E+09,9E+09,9E+09,9E+09,9E+09,9E+09]];
    CONST robtarget Target_2890:=[[130.43,105.636,-28.8],[1,0,0,0],[-1,0,0,1],[9E+09,9E+09,9E+09,9E+09,9E+09,9E+09]];
    CONST robtarget Target_2900:=[[130.085,105.972,-28.8],[1,0,0,0],[-1,0,0,1],[9E+09,9E+09,9E+09,9E+09,9E+09,9E+09]];
    CONST robtarget Target_2910:=[[129.638,106.331,-28.8],[1,0,0,0],[-1,0,0,1],[9E+09,9E+09,9E+09,9E+09,9E+09,9E+09]];
    CONST robtarget Target_2920:=[[129.095,106.692,-28.8],[1,0,0,0],[-1,0,0,1],[9E+09,9E+09,9E+09,9E+09,9E+09,9E+09]];
    CONST robtarget Target_2930:=[[128.461,107.032,-28.8],[1,0,0,0],[-1,0,0,1],[9E+09,9E+09,9E+09,9E+09,9E+09,9E+09]];
    CONST robtarget Target_2940:=[[127.739,107.328,-28.8],[1,0,0,0],[-1,0,0,1],[9E+09,9E+09,9E+09,9E+09,9E+09,9E+09]];
    CONST robtarget Target_2950:=[[126.937,107.555,-28.8],[1,0,0,0],[-1,0,0,1],[9E+09,9E+09,9E+09,9E+09,9E+09,9E+09]];
    CONST robtarget Target_2960:=[[126.097,107.712,-28.8],[1,0,0,0],[-1,0,0,1],[9E+09,9E+09,9E+09,9E+09,9E+09,9E+09]];
    CONST robtarget Target_2970:=[[125.267,107.823,-28.8],[1,0,0,0],[-1,0,0,1],[9E+09,9E+09,9E+09,9E+09,9E+09,9E+09]];
    CONST robtarget Target_2980:=[[124.447,107.887,-28.8],[1,0,0,0],[-1,0,0,1],[9E+09,9E+09,9E+09,9E+09,9E+09,9E+09]];
    CONST robtarget Target_2990:=[[123.631,107.909,-28.8],[1,0,0,0],[-1,0,0,1],[9E+09,9E+09,9E+09,9E+09,9E+09,9E+09]];
    CONST robtarget Target_3000:=[[112.749,107.909,-28.8],[1,0,0,0],[-1,0,0,1],[9E+09,9E+09,9E+09,9E+09,9E+09,9E+09]];
    CONST robtarget Target_3010:=[[112.749,112.075,-28.8],[1,0,0,0],[-1,0,0,1],[9E+09,9E+09,9E+09,9E+09,9E+09,9E+09]];
    CONST robtarget Target_3020:=[[107.601,112.075,-28.8],[1,0,0,0],[-1,0,0,1],[9E+09,9E+09,9E+09,9E+09,9E+09,9E+09]];
    CONST robtarget Target_3030:=[[106.343,108.106,-28.8],[1,0,0,0],[-1,0,0,1],[9E+09,9E+09,9E+09,9E+09,9E+09,9E+09]];
    CONST robtarget Target_3040:=[[99.023,108.075,-28.8],[1,0,0,0],[-1,0,0,1],[9E+09,9E+09,9E+09,9E+09,9E+09,9E+09]];
    CONST robtarget Target_3050:=[[99.023,100.571,-28.8],[1,0,0,0],[-1,0,0,1],[9E+09,9E+09,9E+09,9E+09,9E+09,9E+09]];
    CONST robtarget Target_3060:=[[106.193,100.571,-28.8],[1,0,0,0],[-1,0,0,1],[9E+09,9E+09,9E+09,9E+09,9E+09,9E+09]];
    CONST robtarget Target_3070:=[[106.193,95.236,-28.8],[1,0,0,0],[-1,0,0,1],[9E+09,9E+09,9E+09,9E+09,9E+09,9E+09]];
    CONST robtarget Target_3080:=[[112.641,95.236,-28.8],[1,0,0,0],[-1,0,0,1],[9E+09,9E+09,9E+09,9E+09,9E+09,9E+09]];
    CONST robtarget Target_3090:=[[112.641,100.516,-28.8],[1,0,0,0],[-1,0,0,1],[9E+09,9E+09,9E+09,9E+09,9E+09,9E+09]];
    CONST robtarget Target_3100:=[[123.59,100.516,-28.8],[1,0,0,0],[-1,0,0,1],[9E+09,9E+09,9E+09,9E+09,9E+09,9E+09]];
    CONST robtarget Target_3110:=[[124.004,100.388,-28.8],[1,0,0,0],[-1,0,0,1],[9E+09,9E+09,9E+09,9E+09,9E+09,9E+09]];
    CONST robtarget Target_3120:=[[124.404,100.256,-28.8],[1,0,0,0],[-1,0,0,1],[9E+09,9E+09,9E+09,9E+09,9E+09,9E+09]];
    CONST robtarget Target_3130:=[[124.774,100.077,-28.8],[1,0,0,0],[-1,0,0,1],[9E+09,9E+09,9E+09,9E+09,9E+09,9E+09]];
    CONST robtarget Target_3140:=[[125.099,99.85,-28.8],[1,0,0,0],[-1,0,0,1],[9E+09,9E+09,9E+09,9E+09,9E+09,9E+09]];
    CONST robtarget Target_3150:=[[125.362,99.554,-28.8],[1,0,0,0],[-1,0,0,1],[9E+09,9E+09,9E+09,9E+09,9E+09,9E+09]];
    CONST robtarget Target_3160:=[[125.55,99.172,-28.8],[1,0,0,0],[-1,0,0,1],[9E+09,9E+09,9E+09,9E+09,9E+09,9E+09]];
    CONST robtarget Target_3170:=[[125.647,98.681,-28.8],[1,0,0,0],[-1,0,0,1],[9E+09,9E+09,9E+09,9E+09,9E+09,9E+09]];
    CONST robtarget Target_3180:=[[125.688,98.135,-28.8],[1,0,0,0],[-1,0,0,1],[9E+09,9E+09,9E+09,9E+09,9E+09,9E+09]];
    CONST robtarget Target_3190:=[[125.707,97.592,-28.8],[1,0,0,0],[-1,0,0,1],[9E+09,9E+09,9E+09,9E+09,9E+09,9E+09]];
    CONST robtarget Target_3200:=[[125.713,97.052,-28.8],[1,0,0,0],[-1,0,0,1],[9E+09,9E+09,9E+09,9E+09,9E+09,9E+09]];
    CONST robtarget Target_3210:=[[125.705,96.512,-28.8],[1,0,0,0],[-1,0,0,1],[9E+09,9E+09,9E+09,9E+09,9E+09,9E+09]];
    CONST robtarget Target_3220:=[[125.69,95.975,-28.8],[1,0,0,0],[-1,0,0,1],[9E+09,9E+09,9E+09,9E+09,9E+09,9E+09]];
    CONST robtarget Target_3230:=[[125.649,94.901,-28.8],[1,0,0,0],[-1,0,0,1],[9E+09,9E+09,9E+09,9E+09,9E+09,9E+09]];
    CONST robtarget Target_3239:=[[131.371,114.633,-38.8],[1,0,0,0],[-1,0,0,1],[9E+09,9E+09,9E+09,9E+09,9E+09,9E+09]];
    CONST robtarget Target_3240:=[[131.371,114.633,-28.8],[1,0,0,0],[-1,0,0,1],[9E+09,9E+09,9E+09,9E+09,9E+09,9E+09]];
    CONST robtarget Target_3250:=[[131.371,122.192,-28.8],[1,0,0,0],[-1,0,0,1],[9E+09,9E+09,9E+09,9E+09,9E+09,9E+09]];
    CONST robtarget Target_3260:=[[106.36,122.192,-28.8],[1,0,0,0],[-1,0,0,1],[9E+09,9E+09,9E+09,9E+09,9E+09,9E+09]];
    CONST robtarget Target_3270:=[[106.36,114.633,-28.8],[1,0,0,0],[-1,0,0,1],[9E+09,9E+09,9E+09,9E+09,9E+09,9E+09]];
    CONST robtarget Target_3279:=[[97.562,114.715,-38.8],[1,0,0,0],[-1,0,0,1],[9E+09,9E+09,9E+09,9E+09,9E+09,9E+09]];
    CONST robtarget Target_3280:=[[97.562,114.715,-28.8],[1,0,0,0],[-1,0,0,1],[9E+09,9E+09,9E+09,9E+09,9E+09,9E+09]];
    CONST robtarget Target_3290:=[[98.737,114.283,-28.8],[1,0,0,0],[-1,0,0,1],[9E+09,9E+09,9E+09,9E+09,9E+09,9E+09]];
    CONST robtarget Target_3300:=[[99.826,114.194,-28.8],[1,0,0,0],[-1,0,0,1],[9E+09,9E+09,9E+09,9E+09,9E+09,9E+09]];
    CONST robtarget Target_3310:=[[101.09,114.442,-28.8],[1,0,0,0],[-1,0,0,1],[9E+09,9E+09,9E+09,9E+09,9E+09,9E+09]];
    CONST robtarget Target_3320:=[[102.234,115.057,-28.8],[1,0,0,0],[-1,0,0,1],[9E+09,9E+09,9E+09,9E+09,9E+09,9E+09]];
    CONST robtarget Target_3330:=[[103.293,116.203,-28.8],[1,0,0,0],[-1,0,0,1],[9E+09,9E+09,9E+09,9E+09,9E+09,9E+09]];
    CONST robtarget Target_3340:=[[103.942,118.045,-28.8],[1,0,0,0],[-1,0,0,1],[9E+09,9E+09,9E+09,9E+09,9E+09,9E+09]];
    CONST robtarget Target_3350:=[[103.676,120.091,-28.8],[1,0,0,0],[-1,0,0,1],[9E+09,9E+09,9E+09,9E+09,9E+09,9E+09]];
    CONST robtarget Target_3360:=[[102.871,121.41,-28.8],[1,0,0,0],[-1,0,0,1],[9E+09,9E+09,9E+09,9E+09,9E+09,9E+09]];
    CONST robtarget Target_3370:=[[101.96,122.185,-28.8],[1,0,0,0],[-1,0,0,1],[9E+09,9E+09,9E+09,9E+09,9E+09,9E+09]];
    CONST robtarget Target_3380:=[[101.296,122.531,-28.8],[1,0,0,0],[-1,0,0,1],[9E+09,9E+09,9E+09,9E+09,9E+09,9E+09]];
    CONST robtarget Target_3390:=[[100.028,122.844,-28.8],[1,0,0,0],[-1,0,0,1],[9E+09,9E+09,9E+09,9E+09,9E+09,9E+09]];
    CONST robtarget Target_3400:=[[99.226,122.838,-28.8],[1,0,0,0],[-1,0,0,1],[9E+09,9E+09,9E+09,9E+09,9E+09,9E+09]];
    CONST robtarget Target_3410:=[[98.635,122.738,-28.8],[1,0,0,0],[-1,0,0,1],[9E+09,9E+09,9E+09,9E+09,9E+09,9E+09]];
    CONST robtarget Target_3420:=[[97.812,122.448,-28.8],[1,0,0,0],[-1,0,0,1],[9E+09,9E+09,9E+09,9E+09,9E+09,9E+09]];
    CONST robtarget Target_3430:=[[96.753,121.745,-28.8],[1,0,0,0],[-1,0,0,1],[9E+09,9E+09,9E+09,9E+09,9E+09,9E+09]];
    CONST robtarget Target_3440:=[[96.157,121.087,-28.8],[1,0,0,0],[-1,0,0,1],[9E+09,9E+09,9E+09,9E+09,9E+09,9E+09]];
    CONST robtarget Target_3450:=[[95.509,119.801,-28.8],[1,0,0,0],[-1,0,0,1],[9E+09,9E+09,9E+09,9E+09,9E+09,9E+09]];
    CONST robtarget Target_3460:=[[95.335,118.109,-28.8],[1,0,0,0],[-1,0,0,1],[9E+09,9E+09,9E+09,9E+09,9E+09,9E+09]];
    CONST robtarget Target_3470:=[[95.781,116.563,-28.8],[1,0,0,0],[-1,0,0,1],[9E+09,9E+09,9E+09,9E+09,9E+09,9E+09]];
    CONST robtarget Target_3480:=[[96.614,115.421,-28.8],[1,0,0,0],[-1,0,0,1],[9E+09,9E+09,9E+09,9E+09,9E+09,9E+09]];
    CONST robtarget Target_3489:=[[109.94,126.249,-38.8],[1,0,0,0],[-1,0,0,1],[9E+09,9E+09,9E+09,9E+09,9E+09,9E+09]];
    CONST robtarget Target_3490:=[[109.94,126.249,-28.8],[1,0,0,0],[-1,0,0,1],[9E+09,9E+09,9E+09,9E+09,9E+09,9E+09]];
    CONST robtarget Target_3500:=[[129.34,126.249,-28.8],[1,0,0,0],[-1,0,0,1],[9E+09,9E+09,9E+09,9E+09,9E+09,9E+09]];
    CONST robtarget Target_3510:=[[129.863,127.122,-28.8],[1,0,0,0],[-1,0,0,1],[9E+09,9E+09,9E+09,9E+09,9E+09,9E+09]];
    CONST robtarget Target_3520:=[[130.37,128.033,-28.8],[1,0,0,0],[-1,0,0,1],[9E+09,9E+09,9E+09,9E+09,9E+09,9E+09]];
    CONST robtarget Target_3530:=[[130.839,129.004,-28.8],[1,0,0,0],[-1,0,0,1],[9E+09,9E+09,9E+09,9E+09,9E+09,9E+09]];
    CONST robtarget Target_3540:=[[131.27,130.086,-28.8],[1,0,0,0],[-1,0,0,1],[9E+09,9E+09,9E+09,9E+09,9E+09,9E+09]];
    CONST robtarget Target_3550:=[[131.64,131.289,-28.8],[1,0,0,0],[-1,0,0,1],[9E+09,9E+09,9E+09,9E+09,9E+09,9E+09]];
    CONST robtarget Target_3560:=[[131.939,132.66,-28.8],[1,0,0,0],[-1,0,0,1],[9E+09,9E+09,9E+09,9E+09,9E+09,9E+09]];
    CONST robtarget Target_3570:=[[132.15,134.238,-28.8],[1,0,0,0],[-1,0,0,1],[9E+09,9E+09,9E+09,9E+09,9E+09,9E+09]];
    CONST robtarget Target_3580:=[[132.267,136.154,-28.8],[1,0,0,0],[-1,0,0,1],[9E+09,9E+09,9E+09,9E+09,9E+09,9E+09]];
    CONST robtarget Target_3590:=[[132.24,138.441,-28.8],[1,0,0,0],[-1,0,0,1],[9E+09,9E+09,9E+09,9E+09,9E+09,9E+09]];
    CONST robtarget Target_3600:=[[132.007,140.927,-28.8],[1,0,0,0],[-1,0,0,1],[9E+09,9E+09,9E+09,9E+09,9E+09,9E+09]];
    CONST robtarget Target_3610:=[[131.496,143.454,-28.8],[1,0,0,0],[-1,0,0,1],[9E+09,9E+09,9E+09,9E+09,9E+09,9E+09]];
    CONST robtarget Target_3620:=[[130.637,145.857,-28.8],[1,0,0,0],[-1,0,0,1],[9E+09,9E+09,9E+09,9E+09,9E+09,9E+09]];
    CONST robtarget Target_3630:=[[129.361,147.975,-28.8],[1,0,0,0],[-1,0,0,1],[9E+09,9E+09,9E+09,9E+09,9E+09,9E+09]];
    CONST robtarget Target_3640:=[[127.601,149.64,-28.8],[1,0,0,0],[-1,0,0,1],[9E+09,9E+09,9E+09,9E+09,9E+09,9E+09]];
    CONST robtarget Target_3650:=[[125.475,150.914,-28.8],[1,0,0,0],[-1,0,0,1],[9E+09,9E+09,9E+09,9E+09,9E+09,9E+09]];
    CONST robtarget Target_3660:=[[123.169,151.965,-28.8],[1,0,0,0],[-1,0,0,1],[9E+09,9E+09,9E+09,9E+09,9E+09,9E+09]];
    CONST robtarget Target_3670:=[[120.671,152.734,-28.8],[1,0,0,0],[-1,0,0,1],[9E+09,9E+09,9E+09,9E+09,9E+09,9E+09]];
    CONST robtarget Target_3680:=[[117.971,153.267,-28.8],[1,0,0,0],[-1,0,0,1],[9E+09,9E+09,9E+09,9E+09,9E+09,9E+09]];
    CONST robtarget Target_3690:=[[115.054,153.541,-28.8],[1,0,0,0],[-1,0,0,1],[9E+09,9E+09,9E+09,9E+09,9E+09,9E+09]];
    CONST robtarget Target_3700:=[[111.889,153.572,-28.8],[1,0,0,0],[-1,0,0,1],[9E+09,9E+09,9E+09,9E+09,9E+09,9E+09]];
    CONST robtarget Target_3710:=[[108.528,153.317,-28.8],[1,0,0,0],[-1,0,0,1],[9E+09,9E+09,9E+09,9E+09,9E+09,9E+09]];
    CONST robtarget Target_3720:=[[105.197,152.71,-28.8],[1,0,0,0],[-1,0,0,1],[9E+09,9E+09,9E+09,9E+09,9E+09,9E+09]];
    CONST robtarget Target_3730:=[[102.257,151.735,-28.8],[1,0,0,0],[-1,0,0,1],[9E+09,9E+09,9E+09,9E+09,9E+09,9E+09]];
    CONST robtarget Target_3740:=[[99.685,150.468,-28.8],[1,0,0,0],[-1,0,0,1],[9E+09,9E+09,9E+09,9E+09,9E+09,9E+09]];
    CONST robtarget Target_3750:=[[97.579,149.025,-28.8],[1,0,0,0],[-1,0,0,1],[9E+09,9E+09,9E+09,9E+09,9E+09,9E+09]];
    CONST robtarget Target_3760:=[[95.919,147.453,-28.8],[1,0,0,0],[-1,0,0,1],[9E+09,9E+09,9E+09,9E+09,9E+09,9E+09]];
    CONST robtarget Target_3770:=[[94.761,145.866,-28.8],[1,0,0,0],[-1,0,0,1],[9E+09,9E+09,9E+09,9E+09,9E+09,9E+09]];
    CONST robtarget Target_3780:=[[94.136,144.356,-28.8],[1,0,0,0],[-1,0,0,1],[9E+09,9E+09,9E+09,9E+09,9E+09,9E+09]];
    CONST robtarget Target_3790:=[[93.808,142.85,-28.8],[1,0,0,0],[-1,0,0,1],[9E+09,9E+09,9E+09,9E+09,9E+09,9E+09]];
    CONST robtarget Target_3800:=[[93.547,141.19,-28.8],[1,0,0,0],[-1,0,0,1],[9E+09,9E+09,9E+09,9E+09,9E+09,9E+09]];
    CONST robtarget Target_3810:=[[93.353,139.473,-28.8],[1,0,0,0],[-1,0,0,1],[9E+09,9E+09,9E+09,9E+09,9E+09,9E+09]];
    CONST robtarget Target_3820:=[[93.246,137.737,-28.8],[1,0,0,0],[-1,0,0,1],[9E+09,9E+09,9E+09,9E+09,9E+09,9E+09]];
    CONST robtarget Target_3830:=[[93.212,136.051,-28.8],[1,0,0,0],[-1,0,0,1],[9E+09,9E+09,9E+09,9E+09,9E+09,9E+09]];
    CONST robtarget Target_3840:=[[93.266,134.481,-28.8],[1,0,0,0],[-1,0,0,1],[9E+09,9E+09,9E+09,9E+09,9E+09,9E+09]];
    CONST robtarget Target_3850:=[[93.405,133.094,-28.8],[1,0,0,0],[-1,0,0,1],[9E+09,9E+09,9E+09,9E+09,9E+09,9E+09]];
    CONST robtarget Target_3860:=[[93.617,131.899,-28.8],[1,0,0,0],[-1,0,0,1],[9E+09,9E+09,9E+09,9E+09,9E+09,9E+09]];
    CONST robtarget Target_3870:=[[93.852,130.888,-28.8],[1,0,0,0],[-1,0,0,1],[9E+09,9E+09,9E+09,9E+09,9E+09,9E+09]];
    CONST robtarget Target_3880:=[[94.105,130.031,-28.8],[1,0,0,0],[-1,0,0,1],[9E+09,9E+09,9E+09,9E+09,9E+09,9E+09]];
    CONST robtarget Target_3890:=[[94.371,129.287,-28.8],[1,0,0,0],[-1,0,0,1],[9E+09,9E+09,9E+09,9E+09,9E+09,9E+09]];
    CONST robtarget Target_3900:=[[94.654,128.631,-28.8],[1,0,0,0],[-1,0,0,1],[9E+09,9E+09,9E+09,9E+09,9E+09,9E+09]];
    CONST robtarget Target_3910:=[[94.947,128.037,-28.8],[1,0,0,0],[-1,0,0,1],[9E+09,9E+09,9E+09,9E+09,9E+09,9E+09]];
    CONST robtarget Target_3920:=[[95.244,127.473,-28.8],[1,0,0,0],[-1,0,0,1],[9E+09,9E+09,9E+09,9E+09,9E+09,9E+09]];
    CONST robtarget Target_3930:=[[101.692,129.139,-28.8],[1,0,0,0],[-1,0,0,1],[9E+09,9E+09,9E+09,9E+09,9E+09,9E+09]];
    CONST robtarget Target_3940:=[[101.283,130.786,-28.8],[1,0,0,0],[-1,0,0,1],[9E+09,9E+09,9E+09,9E+09,9E+09,9E+09]];
    CONST robtarget Target_3950:=[[100.938,132.447,-28.8],[1,0,0,0],[-1,0,0,1],[9E+09,9E+09,9E+09,9E+09,9E+09,9E+09]];
    CONST robtarget Target_3960:=[[100.684,134.123,-28.8],[1,0,0,0],[-1,0,0,1],[9E+09,9E+09,9E+09,9E+09,9E+09,9E+09]];
    CONST robtarget Target_3970:=[[100.6,135.838,-28.8],[1,0,0,0],[-1,0,0,1],[9E+09,9E+09,9E+09,9E+09,9E+09,9E+09]];
    CONST robtarget Target_3980:=[[100.74,137.604,-28.8],[1,0,0,0],[-1,0,0,1],[9E+09,9E+09,9E+09,9E+09,9E+09,9E+09]];
    CONST robtarget Target_3990:=[[101.135,139.421,-28.8],[1,0,0,0],[-1,0,0,1],[9E+09,9E+09,9E+09,9E+09,9E+09,9E+09]];
    CONST robtarget Target_4000:=[[101.835,141.352,-28.8],[1,0,0,0],[-1,0,0,1],[9E+09,9E+09,9E+09,9E+09,9E+09,9E+09]];
    CONST robtarget Target_4010:=[[103.06,143.031,-28.8],[1,0,0,0],[-1,0,0,1],[9E+09,9E+09,9E+09,9E+09,9E+09,9E+09]];
    CONST robtarget Target_4020:=[[104.81,144.308,-28.8],[1,0,0,0],[-1,0,0,1],[9E+09,9E+09,9E+09,9E+09,9E+09,9E+09]];
    CONST robtarget Target_4030:=[[106.91,145.214,-28.8],[1,0,0,0],[-1,0,0,1],[9E+09,9E+09,9E+09,9E+09,9E+09,9E+09]];
    CONST robtarget Target_4040:=[[109.22,145.776,-28.8],[1,0,0,0],[-1,0,0,1],[9E+09,9E+09,9E+09,9E+09,9E+09,9E+09]];
    CONST robtarget Target_4050:=[[111.585,146.029,-28.8],[1,0,0,0],[-1,0,0,1],[9E+09,9E+09,9E+09,9E+09,9E+09,9E+09]];
    CONST robtarget Target_4060:=[[113.858,146.017,-28.8],[1,0,0,0],[-1,0,0,1],[9E+09,9E+09,9E+09,9E+09,9E+09,9E+09]];
    CONST robtarget Target_4070:=[[115.864,145.759,-28.8],[1,0,0,0],[-1,0,0,1],[9E+09,9E+09,9E+09,9E+09,9E+09,9E+09]];
    CONST robtarget Target_4080:=[[117.608,145.403,-28.8],[1,0,0,0],[-1,0,0,1],[9E+09,9E+09,9E+09,9E+09,9E+09,9E+09]];
    CONST robtarget Target_4090:=[[119.151,145.025,-28.8],[1,0,0,0],[-1,0,0,1],[9E+09,9E+09,9E+09,9E+09,9E+09,9E+09]];
    CONST robtarget Target_4100:=[[120.509,144.576,-28.8],[1,0,0,0],[-1,0,0,1],[9E+09,9E+09,9E+09,9E+09,9E+09,9E+09]];
    CONST robtarget Target_4110:=[[121.668,144.016,-28.8],[1,0,0,0],[-1,0,0,1],[9E+09,9E+09,9E+09,9E+09,9E+09,9E+09]];
    CONST robtarget Target_4120:=[[122.651,143.299,-28.8],[1,0,0,0],[-1,0,0,1],[9E+09,9E+09,9E+09,9E+09,9E+09,9E+09]];
    CONST robtarget Target_4130:=[[123.436,142.374,-28.8],[1,0,0,0],[-1,0,0,1],[9E+09,9E+09,9E+09,9E+09,9E+09,9E+09]];
    CONST robtarget Target_4140:=[[124.035,141.21,-28.8],[1,0,0,0],[-1,0,0,1],[9E+09,9E+09,9E+09,9E+09,9E+09,9E+09]];
    CONST robtarget Target_4150:=[[124.449,139.935,-28.8],[1,0,0,0],[-1,0,0,1],[9E+09,9E+09,9E+09,9E+09,9E+09,9E+09]];
    CONST robtarget Target_4160:=[[124.709,138.747,-28.8],[1,0,0,0],[-1,0,0,1],[9E+09,9E+09,9E+09,9E+09,9E+09,9E+09]];
    CONST robtarget Target_4170:=[[124.84,137.625,-28.8],[1,0,0,0],[-1,0,0,1],[9E+09,9E+09,9E+09,9E+09,9E+09,9E+09]];
    CONST robtarget Target_4180:=[[124.867,136.555,-28.8],[1,0,0,0],[-1,0,0,1],[9E+09,9E+09,9E+09,9E+09,9E+09,9E+09]];
    CONST robtarget Target_4190:=[[124.817,135.526,-28.8],[1,0,0,0],[-1,0,0,1],[9E+09,9E+09,9E+09,9E+09,9E+09,9E+09]];
    CONST robtarget Target_4200:=[[124.718,134.521,-28.8],[1,0,0,0],[-1,0,0,1],[9E+09,9E+09,9E+09,9E+09,9E+09,9E+09]];
    CONST robtarget Target_4210:=[[124.59,133.53,-28.8],[1,0,0,0],[-1,0,0,1],[9E+09,9E+09,9E+09,9E+09,9E+09,9E+09]];
    CONST robtarget Target_4220:=[[116.859,133.526,-28.8],[1,0,0,0],[-1,0,0,1],[9E+09,9E+09,9E+09,9E+09,9E+09,9E+09]];
    CONST robtarget Target_4230:=[[116.859,138.922,-28.8],[1,0,0,0],[-1,0,0,1],[9E+09,9E+09,9E+09,9E+09,9E+09,9E+09]];
    CONST robtarget Target_4240:=[[109.94,138.809,-28.8],[1,0,0,0],[-1,0,0,1],[9E+09,9E+09,9E+09,9E+09,9E+09,9E+09]];
    CONST robtarget Target_4249:=[[144,185.869,-38.8],[1,0,0,0],[-1,0,0,1],[9E+09,9E+09,9E+09,9E+09,9E+09,9E+09]];
    CONST robtarget Target_4250:=[[144,185.869,-28.8],[1,0,0,0],[-1,0,0,1],[9E+09,9E+09,9E+09,9E+09,9E+09,9E+09]];
    CONST robtarget Target_4260:=[[143.187,183.493,-28.8],[1,0,0,0],[-1,0,0,1],[9E+09,9E+09,9E+09,9E+09,9E+09,9E+09]];
    CONST robtarget Target_4270:=[[142.423,181.689,-28.8],[1,0,0,0],[-1,0,0,1],[9E+09,9E+09,9E+09,9E+09,9E+09,9E+09]];
    CONST robtarget Target_4280:=[[141.62,180.067,-28.8],[1,0,0,0],[-1,0,0,1],[9E+09,9E+09,9E+09,9E+09,9E+09,9E+09]];
    CONST robtarget Target_4290:=[[140.516,178.152,-28.8],[1,0,0,0],[-1,0,0,1],[9E+09,9E+09,9E+09,9E+09,9E+09,9E+09]];
    CONST robtarget Target_4300:=[[139.233,176.253,-28.8],[1,0,0,0],[-1,0,0,1],[9E+09,9E+09,9E+09,9E+09,9E+09,9E+09]];
    CONST robtarget Target_4310:=[[137.775,174.405,-28.8],[1,0,0,0],[-1,0,0,1],[9E+09,9E+09,9E+09,9E+09,9E+09,9E+09]];
    CONST robtarget Target_4320:=[[136.227,172.712,-28.8],[1,0,0,0],[-1,0,0,1],[9E+09,9E+09,9E+09,9E+09,9E+09,9E+09]];
    CONST robtarget Target_4330:=[[134.701,171.26,-28.8],[1,0,0,0],[-1,0,0,1],[9E+09,9E+09,9E+09,9E+09,9E+09,9E+09]];
    CONST robtarget Target_4340:=[[133.19,169.997,-28.8],[1,0,0,0],[-1,0,0,1],[9E+09,9E+09,9E+09,9E+09,9E+09,9E+09]];
    CONST robtarget Target_4350:=[[131.4,168.692,-28.8],[1,0,0,0],[-1,0,0,1],[9E+09,9E+09,9E+09,9E+09,9E+09,9E+09]];
    CONST robtarget Target_4360:=[[129.85,167.707,-28.8],[1,0,0,0],[-1,0,0,1],[9E+09,9E+09,9E+09,9E+09,9E+09,9E+09]];
    CONST robtarget Target_4370:=[[128.257,166.819,-28.8],[1,0,0,0],[-1,0,0,1],[9E+09,9E+09,9E+09,9E+09,9E+09,9E+09]];
    CONST robtarget Target_4380:=[[126.489,165.967,-28.8],[1,0,0,0],[-1,0,0,1],[9E+09,9E+09,9E+09,9E+09,9E+09,9E+09]];
    CONST robtarget Target_4390:=[[124.107,165.023,-28.8],[1,0,0,0],[-1,0,0,1],[9E+09,9E+09,9E+09,9E+09,9E+09,9E+09]];
    CONST robtarget Target_4400:=[[121.867,164.331,-28.8],[1,0,0,0],[-1,0,0,1],[9E+09,9E+09,9E+09,9E+09,9E+09,9E+09]];
    CONST robtarget Target_4410:=[[119.889,163.866,-28.8],[1,0,0,0],[-1,0,0,1],[9E+09,9E+09,9E+09,9E+09,9E+09,9E+09]];
    CONST robtarget Target_4420:=[[117.828,163.521,-28.8],[1,0,0,0],[-1,0,0,1],[9E+09,9E+09,9E+09,9E+09,9E+09,9E+09]];
    CONST robtarget Target_4430:=[[115.894,163.323,-28.8],[1,0,0,0],[-1,0,0,1],[9E+09,9E+09,9E+09,9E+09,9E+09,9E+09]];
    CONST robtarget Target_4440:=[[113.217,163.244,-28.8],[1,0,0,0],[-1,0,0,1],[9E+09,9E+09,9E+09,9E+09,9E+09,9E+09]];
    CONST robtarget Target_4450:=[[110.663,163.381,-28.8],[1,0,0,0],[-1,0,0,1],[9E+09,9E+09,9E+09,9E+09,9E+09,9E+09]];
    CONST robtarget Target_4460:=[[108.096,163.728,-28.8],[1,0,0,0],[-1,0,0,1],[9E+09,9E+09,9E+09,9E+09,9E+09,9E+09]];
    CONST robtarget Target_4470:=[[106.289,164.103,-28.8],[1,0,0,0],[-1,0,0,1],[9E+09,9E+09,9E+09,9E+09,9E+09,9E+09]];
    CONST robtarget Target_4480:=[[104.277,164.653,-28.8],[1,0,0,0],[-1,0,0,1],[9E+09,9E+09,9E+09,9E+09,9E+09,9E+09]];
    CONST robtarget Target_4490:=[[103.156,165.022,-28.8],[1,0,0,0],[-1,0,0,1],[9E+09,9E+09,9E+09,9E+09,9E+09,9E+09]];
    CONST robtarget Target_4500:=[[101.114,165.817,-28.8],[1,0,0,0],[-1,0,0,1],[9E+09,9E+09,9E+09,9E+09,9E+09,9E+09]];
    CONST robtarget Target_4510:=[[99.455,166.587,-28.8],[1,0,0,0],[-1,0,0,1],[9E+09,9E+09,9E+09,9E+09,9E+09,9E+09]];
    CONST robtarget Target_4520:=[[98.13,167.29,-28.8],[1,0,0,0],[-1,0,0,1],[9E+09,9E+09,9E+09,9E+09,9E+09,9E+09]];
    CONST robtarget Target_4530:=[[96.996,167.957,-28.8],[1,0,0,0],[-1,0,0,1],[9E+09,9E+09,9E+09,9E+09,9E+09,9E+09]];
    CONST robtarget Target_4540:=[[95.592,168.874,-28.8],[1,0,0,0],[-1,0,0,1],[9E+09,9E+09,9E+09,9E+09,9E+09,9E+09]];
    CONST robtarget Target_4550:=[[94.115,169.96,-28.8],[1,0,0,0],[-1,0,0,1],[9E+09,9E+09,9E+09,9E+09,9E+09,9E+09]];
    CONST robtarget Target_4560:=[[93.562,170.403,-28.8],[1,0,0,0],[-1,0,0,1],[9E+09,9E+09,9E+09,9E+09,9E+09,9E+09]];
    CONST robtarget Target_4570:=[[92.505,171.307,-28.8],[1,0,0,0],[-1,0,0,1],[9E+09,9E+09,9E+09,9E+09,9E+09,9E+09]];
    CONST robtarget Target_4580:=[[91.419,172.324,-28.8],[1,0,0,0],[-1,0,0,1],[9E+09,9E+09,9E+09,9E+09,9E+09,9E+09]];
    CONST robtarget Target_4590:=[[90.476,173.291,-28.8],[1,0,0,0],[-1,0,0,1],[9E+09,9E+09,9E+09,9E+09,9E+09,9E+09]];
    CONST robtarget Target_4600:=[[89.799,174.039,-28.8],[1,0,0,0],[-1,0,0,1],[9E+09,9E+09,9E+09,9E+09,9E+09,9E+09]];
    CONST robtarget Target_4610:=[[88.826,175.203,-28.8],[1,0,0,0],[-1,0,0,1],[9E+09,9E+09,9E+09,9E+09,9E+09,9E+09]];
    CONST robtarget Target_4620:=[[87.991,176.301,-28.8],[1,0,0,0],[-1,0,0,1],[9E+09,9E+09,9E+09,9E+09,9E+09,9E+09]];
    CONST robtarget Target_4630:=[[87.156,177.507,-28.8],[1,0,0,0],[-1,0,0,1],[9E+09,9E+09,9E+09,9E+09,9E+09,9E+09]];
    CONST robtarget Target_4640:=[[86.33,178.832,-28.8],[1,0,0,0],[-1,0,0,1],[9E+09,9E+09,9E+09,9E+09,9E+09,9E+09]];
    CONST robtarget Target_4650:=[[85.707,179.938,-28.8],[1,0,0,0],[-1,0,0,1],[9E+09,9E+09,9E+09,9E+09,9E+09,9E+09]];
    CONST robtarget Target_4660:=[[84.945,181.453,-28.8],[1,0,0,0],[-1,0,0,1],[9E+09,9E+09,9E+09,9E+09,9E+09,9E+09]];
    CONST robtarget Target_4670:=[[84.209,183.143,-28.8],[1,0,0,0],[-1,0,0,1],[9E+09,9E+09,9E+09,9E+09,9E+09,9E+09]];
    CONST robtarget Target_4680:=[[83.41,185.373,-28.8],[1,0,0,0],[-1,0,0,1],[9E+09,9E+09,9E+09,9E+09,9E+09,9E+09]];
    CONST robtarget Target_4690:=[[82.79,187.617,-28.8],[1,0,0,0],[-1,0,0,1],[9E+09,9E+09,9E+09,9E+09,9E+09,9E+09]];
    CONST robtarget Target_4700:=[[82.431,189.343,-28.8],[1,0,0,0],[-1,0,0,1],[9E+09,9E+09,9E+09,9E+09,9E+09,9E+09]];
    CONST robtarget Target_4710:=[[82.198,190.848,-28.8],[1,0,0,0],[-1,0,0,1],[9E+09,9E+09,9E+09,9E+09,9E+09,9E+09]];
    CONST robtarget Target_4720:=[[82.013,192.68,-28.8],[1,0,0,0],[-1,0,0,1],[9E+09,9E+09,9E+09,9E+09,9E+09,9E+09]];
    CONST robtarget Target_4730:=[[81.937,194.429,-28.8],[1,0,0,0],[-1,0,0,1],[9E+09,9E+09,9E+09,9E+09,9E+09,9E+09]];
    CONST robtarget Target_4740:=[[81.968,196.432,-28.8],[1,0,0,0],[-1,0,0,1],[9E+09,9E+09,9E+09,9E+09,9E+09,9E+09]];
    CONST robtarget Target_4750:=[[82.075,197.935,-28.8],[1,0,0,0],[-1,0,0,1],[9E+09,9E+09,9E+09,9E+09,9E+09,9E+09]];
    CONST robtarget Target_4760:=[[82.236,199.309,-28.8],[1,0,0,0],[-1,0,0,1],[9E+09,9E+09,9E+09,9E+09,9E+09,9E+09]];
    CONST robtarget Target_4770:=[[82.396,200.339,-28.8],[1,0,0,0],[-1,0,0,1],[9E+09,9E+09,9E+09,9E+09,9E+09,9E+09]];
    CONST robtarget Target_4780:=[[82.603,201.42,-28.8],[1,0,0,0],[-1,0,0,1],[9E+09,9E+09,9E+09,9E+09,9E+09,9E+09]];
    CONST robtarget Target_4790:=[[82.84,202.468,-28.8],[1,0,0,0],[-1,0,0,1],[9E+09,9E+09,9E+09,9E+09,9E+09,9E+09]];
    CONST robtarget Target_4800:=[[82.969,202.976,-28.8],[1,0,0,0],[-1,0,0,1],[9E+09,9E+09,9E+09,9E+09,9E+09,9E+09]];
    CONST robtarget Target_4810:=[[83.203,203.819,-28.8],[1,0,0,0],[-1,0,0,1],[9E+09,9E+09,9E+09,9E+09,9E+09,9E+09]];
    CONST robtarget Target_4820:=[[83.557,204.952,-28.8],[1,0,0,0],[-1,0,0,1],[9E+09,9E+09,9E+09,9E+09,9E+09,9E+09]];
    CONST robtarget Target_4830:=[[83.928,206.005,-28.8],[1,0,0,0],[-1,0,0,1],[9E+09,9E+09,9E+09,9E+09,9E+09,9E+09]];
    CONST robtarget Target_4840:=[[84.367,207.119,-28.8],[1,0,0,0],[-1,0,0,1],[9E+09,9E+09,9E+09,9E+09,9E+09,9E+09]];
    CONST robtarget Target_4850:=[[84.799,208.108,-28.8],[1,0,0,0],[-1,0,0,1],[9E+09,9E+09,9E+09,9E+09,9E+09,9E+09]];
    CONST robtarget Target_4860:=[[85.261,209.077,-28.8],[1,0,0,0],[-1,0,0,1],[9E+09,9E+09,9E+09,9E+09,9E+09,9E+09]];
    CONST robtarget Target_4870:=[[85.722,209.965,-28.8],[1,0,0,0],[-1,0,0,1],[9E+09,9E+09,9E+09,9E+09,9E+09,9E+09]];
    CONST robtarget Target_4880:=[[86.11,210.664,-28.8],[1,0,0,0],[-1,0,0,1],[9E+09,9E+09,9E+09,9E+09,9E+09,9E+09]];
    CONST robtarget Target_4890:=[[86.501,211.33,-28.8],[1,0,0,0],[-1,0,0,1],[9E+09,9E+09,9E+09,9E+09,9E+09,9E+09]];
    CONST robtarget Target_4900:=[[86.883,211.946,-28.8],[1,0,0,0],[-1,0,0,1],[9E+09,9E+09,9E+09,9E+09,9E+09,9E+09]];
    CONST robtarget Target_4910:=[[87.378,212.701,-28.8],[1,0,0,0],[-1,0,0,1],[9E+09,9E+09,9E+09,9E+09,9E+09,9E+09]];
    CONST robtarget Target_4920:=[[87.848,213.376,-28.8],[1,0,0,0],[-1,0,0,1],[9E+09,9E+09,9E+09,9E+09,9E+09,9E+09]];
    CONST robtarget Target_4930:=[[88.345,214.053,-28.8],[1,0,0,0],[-1,0,0,1],[9E+09,9E+09,9E+09,9E+09,9E+09,9E+09]];
    CONST robtarget Target_4940:=[[89.004,214.894,-28.8],[1,0,0,0],[-1,0,0,1],[9E+09,9E+09,9E+09,9E+09,9E+09,9E+09]];
    CONST robtarget Target_4950:=[[89.589,215.595,-28.8],[1,0,0,0],[-1,0,0,1],[9E+09,9E+09,9E+09,9E+09,9E+09,9E+09]];
    CONST robtarget Target_4960:=[[90.252,216.342,-28.8],[1,0,0,0],[-1,0,0,1],[9E+09,9E+09,9E+09,9E+09,9E+09,9E+09]];
    CONST robtarget Target_4970:=[[90.946,217.076,-28.8],[1,0,0,0],[-1,0,0,1],[9E+09,9E+09,9E+09,9E+09,9E+09,9E+09]];
    CONST robtarget Target_4980:=[[91.738,217.86,-28.8],[1,0,0,0],[-1,0,0,1],[9E+09,9E+09,9E+09,9E+09,9E+09,9E+09]];
    CONST robtarget Target_4990:=[[92.511,218.574,-28.8],[1,0,0,0],[-1,0,0,1],[9E+09,9E+09,9E+09,9E+09,9E+09,9E+09]];
    CONST robtarget Target_5000:=[[93.488,219.412,-28.8],[1,0,0,0],[-1,0,0,1],[9E+09,9E+09,9E+09,9E+09,9E+09,9E+09]];
    CONST robtarget Target_5010:=[[94.249,220.019,-28.8],[1,0,0,0],[-1,0,0,1],[9E+09,9E+09,9E+09,9E+09,9E+09,9E+09]];
    CONST robtarget Target_5020:=[[94.928,220.529,-28.8],[1,0,0,0],[-1,0,0,1],[9E+09,9E+09,9E+09,9E+09,9E+09,9E+09]];
    CONST robtarget Target_5030:=[[95.69,221.069,-28.8],[1,0,0,0],[-1,0,0,1],[9E+09,9E+09,9E+09,9E+09,9E+09,9E+09]];
    CONST robtarget Target_5040:=[[96.255,221.448,-28.8],[1,0,0,0],[-1,0,0,1],[9E+09,9E+09,9E+09,9E+09,9E+09,9E+09]];
    CONST robtarget Target_5050:=[[96.932,221.879,-28.8],[1,0,0,0],[-1,0,0,1],[9E+09,9E+09,9E+09,9E+09,9E+09,9E+09]];
    CONST robtarget Target_5060:=[[97.848,222.426,-28.8],[1,0,0,0],[-1,0,0,1],[9E+09,9E+09,9E+09,9E+09,9E+09,9E+09]];
    CONST robtarget Target_5070:=[[98.978,223.045,-28.8],[1,0,0,0],[-1,0,0,1],[9E+09,9E+09,9E+09,9E+09,9E+09,9E+09]];
    CONST robtarget Target_5080:=[[99.732,223.425,-28.8],[1,0,0,0],[-1,0,0,1],[9E+09,9E+09,9E+09,9E+09,9E+09,9E+09]];
    CONST robtarget Target_5090:=[[100.693,223.874,-28.8],[1,0,0,0],[-1,0,0,1],[9E+09,9E+09,9E+09,9E+09,9E+09,9E+09]];
    CONST robtarget Target_5100:=[[101.635,224.277,-28.8],[1,0,0,0],[-1,0,0,1],[9E+09,9E+09,9E+09,9E+09,9E+09,9E+09]];
    CONST robtarget Target_5110:=[[102.631,224.665,-28.8],[1,0,0,0],[-1,0,0,1],[9E+09,9E+09,9E+09,9E+09,9E+09,9E+09]];
    CONST robtarget Target_5120:=[[103.793,225.069,-28.8],[1,0,0,0],[-1,0,0,1],[9E+09,9E+09,9E+09,9E+09,9E+09,9E+09]];
    CONST robtarget Target_5130:=[[104.73,225.359,-28.8],[1,0,0,0],[-1,0,0,1],[9E+09,9E+09,9E+09,9E+09,9E+09,9E+09]];
    CONST robtarget Target_5140:=[[105.724,225.632,-28.8],[1,0,0,0],[-1,0,0,1],[9E+09,9E+09,9E+09,9E+09,9E+09,9E+09]];
    CONST robtarget Target_5150:=[[106.823,225.895,-28.8],[1,0,0,0],[-1,0,0,1],[9E+09,9E+09,9E+09,9E+09,9E+09,9E+09]];
    CONST robtarget Target_5160:=[[107.954,226.122,-28.8],[1,0,0,0],[-1,0,0,1],[9E+09,9E+09,9E+09,9E+09,9E+09,9E+09]];
    CONST robtarget Target_5170:=[[109.276,226.334,-28.8],[1,0,0,0],[-1,0,0,1],[9E+09,9E+09,9E+09,9E+09,9E+09,9E+09]];
    CONST robtarget Target_5180:=[[110.729,226.501,-28.8],[1,0,0,0],[-1,0,0,1],[9E+09,9E+09,9E+09,9E+09,9E+09,9E+09]];
    CONST robtarget Target_5190:=[[111.977,226.591,-28.8],[1,0,0,0],[-1,0,0,1],[9E+09,9E+09,9E+09,9E+09,9E+09,9E+09]];
    CONST robtarget Target_5200:=[[113.215,226.631,-28.8],[1,0,0,0],[-1,0,0,1],[9E+09,9E+09,9E+09,9E+09,9E+09,9E+09]];
    CONST robtarget Target_5210:=[[114.666,226.617,-28.8],[1,0,0,0],[-1,0,0,1],[9E+09,9E+09,9E+09,9E+09,9E+09,9E+09]];
    CONST robtarget Target_5220:=[[116.493,226.504,-28.8],[1,0,0,0],[-1,0,0,1],[9E+09,9E+09,9E+09,9E+09,9E+09,9E+09]];
    CONST robtarget Target_5230:=[[118.822,226.206,-28.8],[1,0,0,0],[-1,0,0,1],[9E+09,9E+09,9E+09,9E+09,9E+09,9E+09]];
    CONST robtarget Target_5240:=[[121.188,225.719,-28.8],[1,0,0,0],[-1,0,0,1],[9E+09,9E+09,9E+09,9E+09,9E+09,9E+09]];
    CONST robtarget Target_5250:=[[123.533,225.047,-28.8],[1,0,0,0],[-1,0,0,1],[9E+09,9E+09,9E+09,9E+09,9E+09,9E+09]];
    CONST robtarget Target_5260:=[[126.022,224.111,-28.8],[1,0,0,0],[-1,0,0,1],[9E+09,9E+09,9E+09,9E+09,9E+09,9E+09]];
    CONST robtarget Target_5270:=[[128.198,223.087,-28.8],[1,0,0,0],[-1,0,0,1],[9E+09,9E+09,9E+09,9E+09,9E+09,9E+09]];
    CONST robtarget Target_5280:=[[130.862,221.54,-28.8],[1,0,0,0],[-1,0,0,1],[9E+09,9E+09,9E+09,9E+09,9E+09,9E+09]];
    CONST robtarget Target_5290:=[[133.022,220.009,-28.8],[1,0,0,0],[-1,0,0,1],[9E+09,9E+09,9E+09,9E+09,9E+09,9E+09]];
    CONST robtarget Target_5300:=[[134.29,218.975,-28.8],[1,0,0,0],[-1,0,0,1],[9E+09,9E+09,9E+09,9E+09,9E+09,9E+09]];
    CONST robtarget Target_5310:=[[136.037,217.355,-28.8],[1,0,0,0],[-1,0,0,1],[9E+09,9E+09,9E+09,9E+09,9E+09,9E+09]];
    CONST robtarget Target_5320:=[[137.627,215.644,-28.8],[1,0,0,0],[-1,0,0,1],[9E+09,9E+09,9E+09,9E+09,9E+09,9E+09]];
    CONST robtarget Target_5330:=[[138.77,214.24,-28.8],[1,0,0,0],[-1,0,0,1],[9E+09,9E+09,9E+09,9E+09,9E+09,9E+09]];
    CONST robtarget Target_5340:=[[140.398,211.91,-28.8],[1,0,0,0],[-1,0,0,1],[9E+09,9E+09,9E+09,9E+09,9E+09,9E+09]];
    CONST robtarget Target_5350:=[[141.508,210.019,-28.8],[1,0,0,0],[-1,0,0,1],[9E+09,9E+09,9E+09,9E+09,9E+09,9E+09]];
    CONST robtarget Target_5360:=[[142.412,208.212,-28.8],[1,0,0,0],[-1,0,0,1],[9E+09,9E+09,9E+09,9E+09,9E+09,9E+09]];
    CONST robtarget Target_5370:=[[142.981,206.901,-28.8],[1,0,0,0],[-1,0,0,1],[9E+09,9E+09,9E+09,9E+09,9E+09,9E+09]];
    CONST robtarget Target_5380:=[[143.596,205.263,-28.8],[1,0,0,0],[-1,0,0,1],[9E+09,9E+09,9E+09,9E+09,9E+09,9E+09]];
    CONST robtarget Target_5390:=[[143.902,204.049,-28.8],[1,0,0,0],[-1,0,0,1],[9E+09,9E+09,9E+09,9E+09,9E+09,9E+09]];
    CONST robtarget Target_5400:=[[143.776,203.162,-28.8],[1,0,0,0],[-1,0,0,1],[9E+09,9E+09,9E+09,9E+09,9E+09,9E+09]];
    CONST robtarget Target_5410:=[[143.201,202.597,-28.8],[1,0,0,0],[-1,0,0,1],[9E+09,9E+09,9E+09,9E+09,9E+09,9E+09]];
    CONST robtarget Target_5420:=[[142.436,202.618,-28.8],[1,0,0,0],[-1,0,0,1],[9E+09,9E+09,9E+09,9E+09,9E+09,9E+09]];
    CONST robtarget Target_5430:=[[141.518,202.643,-28.8],[1,0,0,0],[-1,0,0,1],[9E+09,9E+09,9E+09,9E+09,9E+09,9E+09]];
    CONST robtarget Target_5440:=[[140.796,202.662,-28.8],[1,0,0,0],[-1,0,0,1],[9E+09,9E+09,9E+09,9E+09,9E+09,9E+09]];
    CONST robtarget Target_5450:=[[139.898,202.687,-28.8],[1,0,0,0],[-1,0,0,1],[9E+09,9E+09,9E+09,9E+09,9E+09,9E+09]];
    CONST robtarget Target_5460:=[[138.845,202.715,-28.8],[1,0,0,0],[-1,0,0,1],[9E+09,9E+09,9E+09,9E+09,9E+09,9E+09]];
    CONST robtarget Target_5470:=[[138.008,202.738,-28.8],[1,0,0,0],[-1,0,0,1],[9E+09,9E+09,9E+09,9E+09,9E+09,9E+09]];
    CONST robtarget Target_5480:=[[137.231,202.759,-28.8],[1,0,0,0],[-1,0,0,1],[9E+09,9E+09,9E+09,9E+09,9E+09,9E+09]];
    CONST robtarget Target_5490:=[[136.688,202.773,-28.8],[1,0,0,0],[-1,0,0,1],[9E+09,9E+09,9E+09,9E+09,9E+09,9E+09]];
    CONST robtarget Target_5500:=[[136.832,203.669,-28.8],[1,0,0,0],[-1,0,0,1],[9E+09,9E+09,9E+09,9E+09,9E+09,9E+09]];
    CONST robtarget Target_5510:=[[136.988,204.835,-28.8],[1,0,0,0],[-1,0,0,1],[9E+09,9E+09,9E+09,9E+09,9E+09,9E+09]];
    CONST robtarget Target_5520:=[[137.066,205.811,-28.8],[1,0,0,0],[-1,0,0,1],[9E+09,9E+09,9E+09,9E+09,9E+09,9E+09]];
    CONST robtarget Target_5530:=[[137.064,206.757,-28.8],[1,0,0,0],[-1,0,0,1],[9E+09,9E+09,9E+09,9E+09,9E+09,9E+09]];
    CONST robtarget Target_5540:=[[136.99,207.502,-28.8],[1,0,0,0],[-1,0,0,1],[9E+09,9E+09,9E+09,9E+09,9E+09,9E+09]];
    CONST robtarget Target_5550:=[[136.825,208.289,-28.8],[1,0,0,0],[-1,0,0,1],[9E+09,9E+09,9E+09,9E+09,9E+09,9E+09]];
    CONST robtarget Target_5560:=[[136.504,209.207,-28.8],[1,0,0,0],[-1,0,0,1],[9E+09,9E+09,9E+09,9E+09,9E+09,9E+09]];
    CONST robtarget Target_5570:=[[136.071,210.099,-28.8],[1,0,0,0],[-1,0,0,1],[9E+09,9E+09,9E+09,9E+09,9E+09,9E+09]];
    CONST robtarget Target_5580:=[[135.649,210.801,-28.8],[1,0,0,0],[-1,0,0,1],[9E+09,9E+09,9E+09,9E+09,9E+09,9E+09]];
    CONST robtarget Target_5590:=[[135.02,211.636,-28.8],[1,0,0,0],[-1,0,0,1],[9E+09,9E+09,9E+09,9E+09,9E+09,9E+09]];
    CONST robtarget Target_5600:=[[134.431,212.23,-28.8],[1,0,0,0],[-1,0,0,1],[9E+09,9E+09,9E+09,9E+09,9E+09,9E+09]];
    CONST robtarget Target_5610:=[[133.434,212.857,-28.8],[1,0,0,0],[-1,0,0,1],[9E+09,9E+09,9E+09,9E+09,9E+09,9E+09]];
    CONST robtarget Target_5620:=[[132.756,213.051,-28.8],[1,0,0,0],[-1,0,0,1],[9E+09,9E+09,9E+09,9E+09,9E+09,9E+09]];
    CONST robtarget Target_5630:=[[131.986,213.274,-28.8],[1,0,0,0],[-1,0,0,1],[9E+09,9E+09,9E+09,9E+09,9E+09,9E+09]];
    CONST robtarget Target_5640:=[[131.187,213.673,-28.8],[1,0,0,0],[-1,0,0,1],[9E+09,9E+09,9E+09,9E+09,9E+09,9E+09]];
    CONST robtarget Target_5650:=[[130.19,214.388,-28.8],[1,0,0,0],[-1,0,0,1],[9E+09,9E+09,9E+09,9E+09,9E+09,9E+09]];
    CONST robtarget Target_5660:=[[129.454,215.035,-28.8],[1,0,0,0],[-1,0,0,1],[9E+09,9E+09,9E+09,9E+09,9E+09,9E+09]];
    CONST robtarget Target_5670:=[[128.98,215.492,-28.8],[1,0,0,0],[-1,0,0,1],[9E+09,9E+09,9E+09,9E+09,9E+09,9E+09]];
    CONST robtarget Target_5680:=[[128.144,216.468,-28.8],[1,0,0,0],[-1,0,0,1],[9E+09,9E+09,9E+09,9E+09,9E+09,9E+09]];
    CONST robtarget Target_5690:=[[127.644,217.156,-28.8],[1,0,0,0],[-1,0,0,1],[9E+09,9E+09,9E+09,9E+09,9E+09,9E+09]];
    CONST robtarget Target_5700:=[[127.066,217.667,-28.8],[1,0,0,0],[-1,0,0,1],[9E+09,9E+09,9E+09,9E+09,9E+09,9E+09]];
    CONST robtarget Target_5710:=[[126.606,217.376,-28.8],[1,0,0,0],[-1,0,0,1],[9E+09,9E+09,9E+09,9E+09,9E+09,9E+09]];
    CONST robtarget Target_5720:=[[126.464,216.918,-28.8],[1,0,0,0],[-1,0,0,1],[9E+09,9E+09,9E+09,9E+09,9E+09,9E+09]];
    CONST robtarget Target_5730:=[[126.395,216.33,-28.8],[1,0,0,0],[-1,0,0,1],[9E+09,9E+09,9E+09,9E+09,9E+09,9E+09]];
    CONST robtarget Target_5740:=[[126.423,215.541,-28.8],[1,0,0,0],[-1,0,0,1],[9E+09,9E+09,9E+09,9E+09,9E+09,9E+09]];
    CONST robtarget Target_5750:=[[126.59,214.771,-28.8],[1,0,0,0],[-1,0,0,1],[9E+09,9E+09,9E+09,9E+09,9E+09,9E+09]];
    CONST robtarget Target_5760:=[[126.946,214.057,-28.8],[1,0,0,0],[-1,0,0,1],[9E+09,9E+09,9E+09,9E+09,9E+09,9E+09]];
    CONST robtarget Target_5770:=[[127.442,213.468,-28.8],[1,0,0,0],[-1,0,0,1],[9E+09,9E+09,9E+09,9E+09,9E+09,9E+09]];
    CONST robtarget Target_5780:=[[127.891,213.044,-28.8],[1,0,0,0],[-1,0,0,1],[9E+09,9E+09,9E+09,9E+09,9E+09,9E+09]];
    CONST robtarget Target_5790:=[[128.442,212.573,-28.8],[1,0,0,0],[-1,0,0,1],[9E+09,9E+09,9E+09,9E+09,9E+09,9E+09]];
    CONST robtarget Target_5800:=[[128.925,212.184,-28.8],[1,0,0,0],[-1,0,0,1],[9E+09,9E+09,9E+09,9E+09,9E+09,9E+09]];
    CONST robtarget Target_5810:=[[129.466,211.758,-28.8],[1,0,0,0],[-1,0,0,1],[9E+09,9E+09,9E+09,9E+09,9E+09,9E+09]];
    CONST robtarget Target_5820:=[[130.02,211.315,-28.8],[1,0,0,0],[-1,0,0,1],[9E+09,9E+09,9E+09,9E+09,9E+09,9E+09]];
    CONST robtarget Target_5830:=[[130.631,210.799,-28.8],[1,0,0,0],[-1,0,0,1],[9E+09,9E+09,9E+09,9E+09,9E+09,9E+09]];
    CONST robtarget Target_5840:=[[131.282,210.148,-28.8],[1,0,0,0],[-1,0,0,1],[9E+09,9E+09,9E+09,9E+09,9E+09,9E+09]];
    CONST robtarget Target_5850:=[[131.648,209.677,-28.8],[1,0,0,0],[-1,0,0,1],[9E+09,9E+09,9E+09,9E+09,9E+09,9E+09]];
    CONST robtarget Target_5860:=[[131.923,209.234,-28.8],[1,0,0,0],[-1,0,0,1],[9E+09,9E+09,9E+09,9E+09,9E+09,9E+09]];
    CONST robtarget Target_5870:=[[132.14,208.81,-28.8],[1,0,0,0],[-1,0,0,1],[9E+09,9E+09,9E+09,9E+09,9E+09,9E+09]];
    CONST robtarget Target_5880:=[[132.346,208.328,-28.8],[1,0,0,0],[-1,0,0,1],[9E+09,9E+09,9E+09,9E+09,9E+09,9E+09]];
    CONST robtarget Target_5890:=[[132.521,207.84,-28.8],[1,0,0,0],[-1,0,0,1],[9E+09,9E+09,9E+09,9E+09,9E+09,9E+09]];
    CONST robtarget Target_5900:=[[132.678,207.305,-28.8],[1,0,0,0],[-1,0,0,1],[9E+09,9E+09,9E+09,9E+09,9E+09,9E+09]];
    CONST robtarget Target_5910:=[[132.777,206.899,-28.8],[1,0,0,0],[-1,0,0,1],[9E+09,9E+09,9E+09,9E+09,9E+09,9E+09]];
    CONST robtarget Target_5920:=[[132.851,206.539,-28.8],[1,0,0,0],[-1,0,0,1],[9E+09,9E+09,9E+09,9E+09,9E+09,9E+09]];
    CONST robtarget Target_5930:=[[132.95,205.888,-28.8],[1,0,0,0],[-1,0,0,1],[9E+09,9E+09,9E+09,9E+09,9E+09,9E+09]];
    CONST robtarget Target_5940:=[[132.996,205.383,-28.8],[1,0,0,0],[-1,0,0,1],[9E+09,9E+09,9E+09,9E+09,9E+09,9E+09]];
    CONST robtarget Target_5950:=[[133.01,204.93,-28.8],[1,0,0,0],[-1,0,0,1],[9E+09,9E+09,9E+09,9E+09,9E+09,9E+09]];
    CONST robtarget Target_5960:=[[132.986,204.438,-28.8],[1,0,0,0],[-1,0,0,1],[9E+09,9E+09,9E+09,9E+09,9E+09,9E+09]];
    CONST robtarget Target_5970:=[[132.906,203.977,-28.8],[1,0,0,0],[-1,0,0,1],[9E+09,9E+09,9E+09,9E+09,9E+09,9E+09]];
    CONST robtarget Target_5980:=[[132.691,203.433,-28.8],[1,0,0,0],[-1,0,0,1],[9E+09,9E+09,9E+09,9E+09,9E+09,9E+09]];
    CONST robtarget Target_5990:=[[132.369,202.983,-28.8],[1,0,0,0],[-1,0,0,1],[9E+09,9E+09,9E+09,9E+09,9E+09,9E+09]];
    CONST robtarget Target_6000:=[[131.999,202.64,-28.8],[1,0,0,0],[-1,0,0,1],[9E+09,9E+09,9E+09,9E+09,9E+09,9E+09]];
    CONST robtarget Target_6010:=[[131.516,202.342,-28.8],[1,0,0,0],[-1,0,0,1],[9E+09,9E+09,9E+09,9E+09,9E+09,9E+09]];
    CONST robtarget Target_6020:=[[131.022,202.164,-28.8],[1,0,0,0],[-1,0,0,1],[9E+09,9E+09,9E+09,9E+09,9E+09,9E+09]];
    CONST robtarget Target_6030:=[[130.419,202.084,-28.8],[1,0,0,0],[-1,0,0,1],[9E+09,9E+09,9E+09,9E+09,9E+09,9E+09]];
    CONST robtarget Target_6040:=[[129.876,201.914,-28.8],[1,0,0,0],[-1,0,0,1],[9E+09,9E+09,9E+09,9E+09,9E+09,9E+09]];
    CONST robtarget Target_6050:=[[129.431,201.691,-28.8],[1,0,0,0],[-1,0,0,1],[9E+09,9E+09,9E+09,9E+09,9E+09,9E+09]];
    CONST robtarget Target_6060:=[[128.939,201.4,-28.8],[1,0,0,0],[-1,0,0,1],[9E+09,9E+09,9E+09,9E+09,9E+09,9E+09]];
    CONST robtarget Target_6070:=[[128.49,201.113,-28.8],[1,0,0,0],[-1,0,0,1],[9E+09,9E+09,9E+09,9E+09,9E+09,9E+09]];
    CONST robtarget Target_6080:=[[128.135,200.877,-28.8],[1,0,0,0],[-1,0,0,1],[9E+09,9E+09,9E+09,9E+09,9E+09,9E+09]];
    CONST robtarget Target_6090:=[[127.83,200.672,-28.8],[1,0,0,0],[-1,0,0,1],[9E+09,9E+09,9E+09,9E+09,9E+09,9E+09]];
    CONST robtarget Target_6100:=[[127.756,201.176,-28.8],[1,0,0,0],[-1,0,0,1],[9E+09,9E+09,9E+09,9E+09,9E+09,9E+09]];
    CONST robtarget Target_6110:=[[127.672,201.747,-28.8],[1,0,0,0],[-1,0,0,1],[9E+09,9E+09,9E+09,9E+09,9E+09,9E+09]];
    CONST robtarget Target_6120:=[[127.582,202.345,-28.8],[1,0,0,0],[-1,0,0,1],[9E+09,9E+09,9E+09,9E+09,9E+09,9E+09]];
    CONST robtarget Target_6130:=[[127.469,203.055,-28.8],[1,0,0,0],[-1,0,0,1],[9E+09,9E+09,9E+09,9E+09,9E+09,9E+09]];
    CONST robtarget Target_6140:=[[127.338,203.818,-28.8],[1,0,0,0],[-1,0,0,1],[9E+09,9E+09,9E+09,9E+09,9E+09,9E+09]];
    CONST robtarget Target_6150:=[[127.176,204.672,-28.8],[1,0,0,0],[-1,0,0,1],[9E+09,9E+09,9E+09,9E+09,9E+09,9E+09]];
    CONST robtarget Target_6160:=[[127.004,205.453,-28.8],[1,0,0,0],[-1,0,0,1],[9E+09,9E+09,9E+09,9E+09,9E+09,9E+09]];
    CONST robtarget Target_6170:=[[126.809,206.191,-28.8],[1,0,0,0],[-1,0,0,1],[9E+09,9E+09,9E+09,9E+09,9E+09,9E+09]];
    CONST robtarget Target_6180:=[[126.576,206.861,-28.8],[1,0,0,0],[-1,0,0,1],[9E+09,9E+09,9E+09,9E+09,9E+09,9E+09]];
    CONST robtarget Target_6190:=[[126.276,207.53,-28.8],[1,0,0,0],[-1,0,0,1],[9E+09,9E+09,9E+09,9E+09,9E+09,9E+09]];
    CONST robtarget Target_6200:=[[125.818,208.307,-28.8],[1,0,0,0],[-1,0,0,1],[9E+09,9E+09,9E+09,9E+09,9E+09,9E+09]];
    CONST robtarget Target_6210:=[[125.418,208.894,-28.8],[1,0,0,0],[-1,0,0,1],[9E+09,9E+09,9E+09,9E+09,9E+09,9E+09]];
    CONST robtarget Target_6220:=[[124.991,209.468,-28.8],[1,0,0,0],[-1,0,0,1],[9E+09,9E+09,9E+09,9E+09,9E+09,9E+09]];
    CONST robtarget Target_6230:=[[124.37,210.218,-28.8],[1,0,0,0],[-1,0,0,1],[9E+09,9E+09,9E+09,9E+09,9E+09,9E+09]];
    CONST robtarget Target_6240:=[[123.831,210.798,-28.8],[1,0,0,0],[-1,0,0,1],[9E+09,9E+09,9E+09,9E+09,9E+09,9E+09]];
    CONST robtarget Target_6250:=[[123.198,211.403,-28.8],[1,0,0,0],[-1,0,0,1],[9E+09,9E+09,9E+09,9E+09,9E+09,9E+09]];
    CONST robtarget Target_6260:=[[122.544,211.951,-28.8],[1,0,0,0],[-1,0,0,1],[9E+09,9E+09,9E+09,9E+09,9E+09,9E+09]];
    CONST robtarget Target_6270:=[[121.888,212.43,-28.8],[1,0,0,0],[-1,0,0,1],[9E+09,9E+09,9E+09,9E+09,9E+09,9E+09]];
    CONST robtarget Target_6280:=[[121.325,212.789,-28.8],[1,0,0,0],[-1,0,0,1],[9E+09,9E+09,9E+09,9E+09,9E+09,9E+09]];
    CONST robtarget Target_6290:=[[120.925,213.016,-28.8],[1,0,0,0],[-1,0,0,1],[9E+09,9E+09,9E+09,9E+09,9E+09,9E+09]];
    CONST robtarget Target_6300:=[[120.542,213.213,-28.8],[1,0,0,0],[-1,0,0,1],[9E+09,9E+09,9E+09,9E+09,9E+09,9E+09]];
    CONST robtarget Target_6310:=[[119.965,213.474,-28.8],[1,0,0,0],[-1,0,0,1],[9E+09,9E+09,9E+09,9E+09,9E+09,9E+09]];
    CONST robtarget Target_6320:=[[119.515,213.651,-28.8],[1,0,0,0],[-1,0,0,1],[9E+09,9E+09,9E+09,9E+09,9E+09,9E+09]];
    CONST robtarget Target_6330:=[[118.803,213.889,-28.8],[1,0,0,0],[-1,0,0,1],[9E+09,9E+09,9E+09,9E+09,9E+09,9E+09]];
    CONST robtarget Target_6340:=[[118.254,214.043,-28.8],[1,0,0,0],[-1,0,0,1],[9E+09,9E+09,9E+09,9E+09,9E+09,9E+09]];
    CONST robtarget Target_6350:=[[117.69,214.179,-28.8],[1,0,0,0],[-1,0,0,1],[9E+09,9E+09,9E+09,9E+09,9E+09,9E+09]];
    CONST robtarget Target_6360:=[[117.181,214.286,-28.8],[1,0,0,0],[-1,0,0,1],[9E+09,9E+09,9E+09,9E+09,9E+09,9E+09]];
    CONST robtarget Target_6370:=[[116.625,214.389,-28.8],[1,0,0,0],[-1,0,0,1],[9E+09,9E+09,9E+09,9E+09,9E+09,9E+09]];
    CONST robtarget Target_6380:=[[116.019,214.487,-28.8],[1,0,0,0],[-1,0,0,1],[9E+09,9E+09,9E+09,9E+09,9E+09,9E+09]];
    CONST robtarget Target_6390:=[[115.328,214.585,-28.8],[1,0,0,0],[-1,0,0,1],[9E+09,9E+09,9E+09,9E+09,9E+09,9E+09]];
    CONST robtarget Target_6400:=[[114.628,214.668,-28.8],[1,0,0,0],[-1,0,0,1],[9E+09,9E+09,9E+09,9E+09,9E+09,9E+09]];
    CONST robtarget Target_6410:=[[113.831,214.739,-28.8],[1,0,0,0],[-1,0,0,1],[9E+09,9E+09,9E+09,9E+09,9E+09,9E+09]];
    CONST robtarget Target_6420:=[[112.679,214.792,-28.8],[1,0,0,0],[-1,0,0,1],[9E+09,9E+09,9E+09,9E+09,9E+09,9E+09]];
    CONST robtarget Target_6430:=[[111.791,214.782,-28.8],[1,0,0,0],[-1,0,0,1],[9E+09,9E+09,9E+09,9E+09,9E+09,9E+09]];
    CONST robtarget Target_6440:=[[110.553,214.673,-28.8],[1,0,0,0],[-1,0,0,1],[9E+09,9E+09,9E+09,9E+09,9E+09,9E+09]];
    CONST robtarget Target_6450:=[[109.079,214.363,-28.8],[1,0,0,0],[-1,0,0,1],[9E+09,9E+09,9E+09,9E+09,9E+09,9E+09]];
    CONST robtarget Target_6460:=[[107.965,213.978,-28.8],[1,0,0,0],[-1,0,0,1],[9E+09,9E+09,9E+09,9E+09,9E+09,9E+09]];
    CONST robtarget Target_6470:=[[106.642,213.378,-28.8],[1,0,0,0],[-1,0,0,1],[9E+09,9E+09,9E+09,9E+09,9E+09,9E+09]];
    CONST robtarget Target_6480:=[[105.597,212.831,-28.8],[1,0,0,0],[-1,0,0,1],[9E+09,9E+09,9E+09,9E+09,9E+09,9E+09]];
    CONST robtarget Target_6490:=[[104.547,212.237,-28.8],[1,0,0,0],[-1,0,0,1],[9E+09,9E+09,9E+09,9E+09,9E+09,9E+09]];
    CONST robtarget Target_6500:=[[103.32,211.526,-28.8],[1,0,0,0],[-1,0,0,1],[9E+09,9E+09,9E+09,9E+09,9E+09,9E+09]];
    CONST robtarget Target_6510:=[[102.284,211.712,-28.8],[1,0,0,0],[-1,0,0,1],[9E+09,9E+09,9E+09,9E+09,9E+09,9E+09]];
    CONST robtarget Target_6520:=[[101.279,211.916,-28.8],[1,0,0,0],[-1,0,0,1],[9E+09,9E+09,9E+09,9E+09,9E+09,9E+09]];
    CONST robtarget Target_6530:=[[99.994,212.07,-28.8],[1,0,0,0],[-1,0,0,1],[9E+09,9E+09,9E+09,9E+09,9E+09,9E+09]];
    CONST robtarget Target_6540:=[[98.812,212.029,-28.8],[1,0,0,0],[-1,0,0,1],[9E+09,9E+09,9E+09,9E+09,9E+09,9E+09]];
    CONST robtarget Target_6550:=[[97.713,211.859,-28.8],[1,0,0,0],[-1,0,0,1],[9E+09,9E+09,9E+09,9E+09,9E+09,9E+09]];
    CONST robtarget Target_6560:=[[96.789,211.657,-28.8],[1,0,0,0],[-1,0,0,1],[9E+09,9E+09,9E+09,9E+09,9E+09,9E+09]];
    CONST robtarget Target_6570:=[[95.935,211.441,-28.8],[1,0,0,0],[-1,0,0,1],[9E+09,9E+09,9E+09,9E+09,9E+09,9E+09]];
    CONST robtarget Target_6580:=[[94.844,211.057,-28.8],[1,0,0,0],[-1,0,0,1],[9E+09,9E+09,9E+09,9E+09,9E+09,9E+09]];
    CONST robtarget Target_6590:=[[94.956,209.194,-28.8],[1,0,0,0],[-1,0,0,1],[9E+09,9E+09,9E+09,9E+09,9E+09,9E+09]];
    CONST robtarget Target_6600:=[[95.388,207.677,-28.8],[1,0,0,0],[-1,0,0,1],[9E+09,9E+09,9E+09,9E+09,9E+09,9E+09]];
    CONST robtarget Target_6610:=[[96.276,205.741,-28.8],[1,0,0,0],[-1,0,0,1],[9E+09,9E+09,9E+09,9E+09,9E+09,9E+09]];
    CONST robtarget Target_6620:=[[97.324,204.037,-28.8],[1,0,0,0],[-1,0,0,1],[9E+09,9E+09,9E+09,9E+09,9E+09,9E+09]];
    CONST robtarget Target_6630:=[[98.207,202.763,-28.8],[1,0,0,0],[-1,0,0,1],[9E+09,9E+09,9E+09,9E+09,9E+09,9E+09]];
    CONST robtarget Target_6640:=[[97.902,201.521,-28.8],[1,0,0,0],[-1,0,0,1],[9E+09,9E+09,9E+09,9E+09,9E+09,9E+09]];
    CONST robtarget Target_6650:=[[97.638,200.324,-28.8],[1,0,0,0],[-1,0,0,1],[9E+09,9E+09,9E+09,9E+09,9E+09,9E+09]];
    CONST robtarget Target_6660:=[[97.421,199.137,-28.8],[1,0,0,0],[-1,0,0,1],[9E+09,9E+09,9E+09,9E+09,9E+09,9E+09]];
    CONST robtarget Target_6670:=[[97.287,198.128,-28.8],[1,0,0,0],[-1,0,0,1],[9E+09,9E+09,9E+09,9E+09,9E+09,9E+09]];
    CONST robtarget Target_6680:=[[97.188,197.02,-28.8],[1,0,0,0],[-1,0,0,1],[9E+09,9E+09,9E+09,9E+09,9E+09,9E+09]];
    CONST robtarget Target_6690:=[[97.144,196.227,-28.8],[1,0,0,0],[-1,0,0,1],[9E+09,9E+09,9E+09,9E+09,9E+09,9E+09]];
    CONST robtarget Target_6700:=[[97.139,194.944,-28.8],[1,0,0,0],[-1,0,0,1],[9E+09,9E+09,9E+09,9E+09,9E+09,9E+09]];
    CONST robtarget Target_6710:=[[97.18,193.898,-28.8],[1,0,0,0],[-1,0,0,1],[9E+09,9E+09,9E+09,9E+09,9E+09,9E+09]];
    CONST robtarget Target_6720:=[[97.277,192.525,-28.8],[1,0,0,0],[-1,0,0,1],[9E+09,9E+09,9E+09,9E+09,9E+09,9E+09]];
    CONST robtarget Target_6730:=[[97.375,191.556,-28.8],[1,0,0,0],[-1,0,0,1],[9E+09,9E+09,9E+09,9E+09,9E+09,9E+09]];
    CONST robtarget Target_6740:=[[97.464,190.86,-28.8],[1,0,0,0],[-1,0,0,1],[9E+09,9E+09,9E+09,9E+09,9E+09,9E+09]];
    CONST robtarget Target_6750:=[[97.617,189.905,-28.8],[1,0,0,0],[-1,0,0,1],[9E+09,9E+09,9E+09,9E+09,9E+09,9E+09]];
    CONST robtarget Target_6760:=[[97.883,188.603,-28.8],[1,0,0,0],[-1,0,0,1],[9E+09,9E+09,9E+09,9E+09,9E+09,9E+09]];
    CONST robtarget Target_6770:=[[98.136,187.546,-28.8],[1,0,0,0],[-1,0,0,1],[9E+09,9E+09,9E+09,9E+09,9E+09,9E+09]];
    CONST robtarget Target_6780:=[[98.27,186.942,-28.8],[1,0,0,0],[-1,0,0,1],[9E+09,9E+09,9E+09,9E+09,9E+09,9E+09]];
    CONST robtarget Target_6790:=[[97.913,186.436,-28.8],[1,0,0,0],[-1,0,0,1],[9E+09,9E+09,9E+09,9E+09,9E+09,9E+09]];
    CONST robtarget Target_6800:=[[97.456,185.77,-28.8],[1,0,0,0],[-1,0,0,1],[9E+09,9E+09,9E+09,9E+09,9E+09,9E+09]];
    CONST robtarget Target_6810:=[[96.978,185.037,-28.8],[1,0,0,0],[-1,0,0,1],[9E+09,9E+09,9E+09,9E+09,9E+09,9E+09]];
    CONST robtarget Target_6820:=[[96.333,183.946,-28.8],[1,0,0,0],[-1,0,0,1],[9E+09,9E+09,9E+09,9E+09,9E+09,9E+09]];
    CONST robtarget Target_6830:=[[95.871,183.038,-28.8],[1,0,0,0],[-1,0,0,1],[9E+09,9E+09,9E+09,9E+09,9E+09,9E+09]];
    CONST robtarget Target_6840:=[[95.464,182.043,-28.8],[1,0,0,0],[-1,0,0,1],[9E+09,9E+09,9E+09,9E+09,9E+09,9E+09]];
    CONST robtarget Target_6850:=[[95.098,180.779,-28.8],[1,0,0,0],[-1,0,0,1],[9E+09,9E+09,9E+09,9E+09,9E+09,9E+09]];
    CONST robtarget Target_6860:=[[94.914,179.764,-28.8],[1,0,0,0],[-1,0,0,1],[9E+09,9E+09,9E+09,9E+09,9E+09,9E+09]];
    CONST robtarget Target_6870:=[[94.936,178.574,-28.8],[1,0,0,0],[-1,0,0,1],[9E+09,9E+09,9E+09,9E+09,9E+09,9E+09]];
    CONST robtarget Target_6880:=[[96.084,178.266,-28.8],[1,0,0,0],[-1,0,0,1],[9E+09,9E+09,9E+09,9E+09,9E+09,9E+09]];
    CONST robtarget Target_6890:=[[97.19,177.994,-28.8],[1,0,0,0],[-1,0,0,1],[9E+09,9E+09,9E+09,9E+09,9E+09,9E+09]];
    CONST robtarget Target_6900:=[[98.144,177.802,-28.8],[1,0,0,0],[-1,0,0,1],[9E+09,9E+09,9E+09,9E+09,9E+09,9E+09]];
    CONST robtarget Target_6910:=[[98.985,177.687,-28.8],[1,0,0,0],[-1,0,0,1],[9E+09,9E+09,9E+09,9E+09,9E+09,9E+09]];
    CONST robtarget Target_6920:=[[99.978,177.651,-28.8],[1,0,0,0],[-1,0,0,1],[9E+09,9E+09,9E+09,9E+09,9E+09,9E+09]];
    CONST robtarget Target_6930:=[[100.993,177.751,-28.8],[1,0,0,0],[-1,0,0,1],[9E+09,9E+09,9E+09,9E+09,9E+09,9E+09]];
    CONST robtarget Target_6940:=[[101.901,177.915,-28.8],[1,0,0,0],[-1,0,0,1],[9E+09,9E+09,9E+09,9E+09,9E+09,9E+09]];
    CONST robtarget Target_6950:=[[102.555,178.056,-28.8],[1,0,0,0],[-1,0,0,1],[9E+09,9E+09,9E+09,9E+09,9E+09,9E+09]];
    CONST robtarget Target_6960:=[[103.398,178.2,-28.8],[1,0,0,0],[-1,0,0,1],[9E+09,9E+09,9E+09,9E+09,9E+09,9E+09]];
    CONST robtarget Target_6970:=[[103.991,178.17,-28.8],[1,0,0,0],[-1,0,0,1],[9E+09,9E+09,9E+09,9E+09,9E+09,9E+09]];
    CONST robtarget Target_6980:=[[104.579,177.852,-28.8],[1,0,0,0],[-1,0,0,1],[9E+09,9E+09,9E+09,9E+09,9E+09,9E+09]];
    CONST robtarget Target_6990:=[[105.242,177.469,-28.8],[1,0,0,0],[-1,0,0,1],[9E+09,9E+09,9E+09,9E+09,9E+09,9E+09]];
    CONST robtarget Target_7000:=[[106.14,176.974,-28.8],[1,0,0,0],[-1,0,0,1],[9E+09,9E+09,9E+09,9E+09,9E+09,9E+09]];
    CONST robtarget Target_7010:=[[107.068,176.499,-28.8],[1,0,0,0],[-1,0,0,1],[9E+09,9E+09,9E+09,9E+09,9E+09,9E+09]];
    CONST robtarget Target_7020:=[[107.817,176.154,-28.8],[1,0,0,0],[-1,0,0,1],[9E+09,9E+09,9E+09,9E+09,9E+09,9E+09]];
    CONST robtarget Target_7030:=[[108.975,175.712,-28.8],[1,0,0,0],[-1,0,0,1],[9E+09,9E+09,9E+09,9E+09,9E+09,9E+09]];
    CONST robtarget Target_7040:=[[109.975,175.443,-28.8],[1,0,0,0],[-1,0,0,1],[9E+09,9E+09,9E+09,9E+09,9E+09,9E+09]];
    CONST robtarget Target_7050:=[[110.856,175.29,-28.8],[1,0,0,0],[-1,0,0,1],[9E+09,9E+09,9E+09,9E+09,9E+09,9E+09]];
    CONST robtarget Target_7060:=[[111.863,175.198,-28.8],[1,0,0,0],[-1,0,0,1],[9E+09,9E+09,9E+09,9E+09,9E+09,9E+09]];
    CONST robtarget Target_7070:=[[112.776,175.178,-28.8],[1,0,0,0],[-1,0,0,1],[9E+09,9E+09,9E+09,9E+09,9E+09,9E+09]];
    CONST robtarget Target_7080:=[[113.691,175.208,-28.8],[1,0,0,0],[-1,0,0,1],[9E+09,9E+09,9E+09,9E+09,9E+09,9E+09]];
    CONST robtarget Target_7090:=[[114.484,175.267,-28.8],[1,0,0,0],[-1,0,0,1],[9E+09,9E+09,9E+09,9E+09,9E+09,9E+09]];
    CONST robtarget Target_7100:=[[115.352,175.361,-28.8],[1,0,0,0],[-1,0,0,1],[9E+09,9E+09,9E+09,9E+09,9E+09,9E+09]];
    CONST robtarget Target_7110:=[[116.207,175.478,-28.8],[1,0,0,0],[-1,0,0,1],[9E+09,9E+09,9E+09,9E+09,9E+09,9E+09]];
    CONST robtarget Target_7120:=[[116.653,175.548,-28.8],[1,0,0,0],[-1,0,0,1],[9E+09,9E+09,9E+09,9E+09,9E+09,9E+09]];
    CONST robtarget Target_7130:=[[117.364,175.676,-28.8],[1,0,0,0],[-1,0,0,1],[9E+09,9E+09,9E+09,9E+09,9E+09,9E+09]];
    CONST robtarget Target_7140:=[[118.22,175.862,-28.8],[1,0,0,0],[-1,0,0,1],[9E+09,9E+09,9E+09,9E+09,9E+09,9E+09]];
    CONST robtarget Target_7150:=[[118.951,176.057,-28.8],[1,0,0,0],[-1,0,0,1],[9E+09,9E+09,9E+09,9E+09,9E+09,9E+09]];
    CONST robtarget Target_7160:=[[119.6,176.267,-28.8],[1,0,0,0],[-1,0,0,1],[9E+09,9E+09,9E+09,9E+09,9E+09,9E+09]];
    CONST robtarget Target_7170:=[[120.244,176.517,-28.8],[1,0,0,0],[-1,0,0,1],[9E+09,9E+09,9E+09,9E+09,9E+09,9E+09]];
    CONST robtarget Target_7180:=[[120.832,176.787,-28.8],[1,0,0,0],[-1,0,0,1],[9E+09,9E+09,9E+09,9E+09,9E+09,9E+09]];
    CONST robtarget Target_7190:=[[121.585,177.199,-28.8],[1,0,0,0],[-1,0,0,1],[9E+09,9E+09,9E+09,9E+09,9E+09,9E+09]];
    CONST robtarget Target_7200:=[[122.166,177.572,-28.8],[1,0,0,0],[-1,0,0,1],[9E+09,9E+09,9E+09,9E+09,9E+09,9E+09]];
    CONST robtarget Target_7210:=[[122.837,178.067,-28.8],[1,0,0,0],[-1,0,0,1],[9E+09,9E+09,9E+09,9E+09,9E+09,9E+09]];
    CONST robtarget Target_7220:=[[123.554,178.68,-28.8],[1,0,0,0],[-1,0,0,1],[9E+09,9E+09,9E+09,9E+09,9E+09,9E+09]];
    CONST robtarget Target_7230:=[[123.957,179.066,-28.8],[1,0,0,0],[-1,0,0,1],[9E+09,9E+09,9E+09,9E+09,9E+09,9E+09]];
    CONST robtarget Target_7240:=[[124.501,179.639,-28.8],[1,0,0,0],[-1,0,0,1],[9E+09,9E+09,9E+09,9E+09,9E+09,9E+09]];
    CONST robtarget Target_7250:=[[125.016,180.241,-28.8],[1,0,0,0],[-1,0,0,1],[9E+09,9E+09,9E+09,9E+09,9E+09,9E+09]];
    CONST robtarget Target_7260:=[[125.43,180.773,-28.8],[1,0,0,0],[-1,0,0,1],[9E+09,9E+09,9E+09,9E+09,9E+09,9E+09]];
    CONST robtarget Target_7270:=[[125.882,181.41,-28.8],[1,0,0,0],[-1,0,0,1],[9E+09,9E+09,9E+09,9E+09,9E+09,9E+09]];
    CONST robtarget Target_7280:=[[126.315,182.092,-28.8],[1,0,0,0],[-1,0,0,1],[9E+09,9E+09,9E+09,9E+09,9E+09,9E+09]];
    CONST robtarget Target_7290:=[[126.716,182.88,-28.8],[1,0,0,0],[-1,0,0,1],[9E+09,9E+09,9E+09,9E+09,9E+09,9E+09]];
    CONST robtarget Target_7300:=[[126.977,183.576,-28.8],[1,0,0,0],[-1,0,0,1],[9E+09,9E+09,9E+09,9E+09,9E+09,9E+09]];
    CONST robtarget Target_7310:=[[127.154,184.18,-28.8],[1,0,0,0],[-1,0,0,1],[9E+09,9E+09,9E+09,9E+09,9E+09,9E+09]];
    CONST robtarget Target_7320:=[[127.4,185.253,-28.8],[1,0,0,0],[-1,0,0,1],[9E+09,9E+09,9E+09,9E+09,9E+09,9E+09]];
    CONST robtarget Target_7330:=[[127.533,185.94,-28.8],[1,0,0,0],[-1,0,0,1],[9E+09,9E+09,9E+09,9E+09,9E+09,9E+09]];
    CONST robtarget Target_7340:=[[127.735,187.118,-28.8],[1,0,0,0],[-1,0,0,1],[9E+09,9E+09,9E+09,9E+09,9E+09,9E+09]];
    CONST robtarget Target_7350:=[[127.834,187.749,-28.8],[1,0,0,0],[-1,0,0,1],[9E+09,9E+09,9E+09,9E+09,9E+09,9E+09]];
    CONST robtarget Target_7360:=[[127.928,188.375,-28.8],[1,0,0,0],[-1,0,0,1],[9E+09,9E+09,9E+09,9E+09,9E+09,9E+09]];
    CONST robtarget Target_7370:=[[128.038,188.997,-28.8],[1,0,0,0],[-1,0,0,1],[9E+09,9E+09,9E+09,9E+09,9E+09,9E+09]];
    CONST robtarget Target_7380:=[[128.485,188.564,-28.8],[1,0,0,0],[-1,0,0,1],[9E+09,9E+09,9E+09,9E+09,9E+09,9E+09]];
    CONST robtarget Target_7390:=[[129.06,188.095,-28.8],[1,0,0,0],[-1,0,0,1],[9E+09,9E+09,9E+09,9E+09,9E+09,9E+09]];
    CONST robtarget Target_7400:=[[129.713,187.692,-28.8],[1,0,0,0],[-1,0,0,1],[9E+09,9E+09,9E+09,9E+09,9E+09,9E+09]];
    CONST robtarget Target_7410:=[[130.415,187.398,-28.8],[1,0,0,0],[-1,0,0,1],[9E+09,9E+09,9E+09,9E+09,9E+09,9E+09]];
    CONST robtarget Target_7420:=[[130.898,187.262,-28.8],[1,0,0,0],[-1,0,0,1],[9E+09,9E+09,9E+09,9E+09,9E+09,9E+09]];
    CONST robtarget Target_7430:=[[131.925,187.092,-28.8],[1,0,0,0],[-1,0,0,1],[9E+09,9E+09,9E+09,9E+09,9E+09,9E+09]];
    CONST robtarget Target_7440:=[[132.779,187.047,-28.8],[1,0,0,0],[-1,0,0,1],[9E+09,9E+09,9E+09,9E+09,9E+09,9E+09]];
    CONST robtarget Target_7450:=[[133.766,187.029,-28.8],[1,0,0,0],[-1,0,0,1],[9E+09,9E+09,9E+09,9E+09,9E+09,9E+09]];
    CONST robtarget Target_7460:=[[134.85,187.019,-28.8],[1,0,0,0],[-1,0,0,1],[9E+09,9E+09,9E+09,9E+09,9E+09,9E+09]];
    CONST robtarget Target_7470:=[[135.832,187.014,-28.8],[1,0,0,0],[-1,0,0,1],[9E+09,9E+09,9E+09,9E+09,9E+09,9E+09]];
    CONST robtarget Target_7480:=[[137.309,187.009,-28.8],[1,0,0,0],[-1,0,0,1],[9E+09,9E+09,9E+09,9E+09,9E+09,9E+09]];
    CONST robtarget Target_7490:=[[139.004,187.006,-28.8],[1,0,0,0],[-1,0,0,1],[9E+09,9E+09,9E+09,9E+09,9E+09,9E+09]];
    CONST robtarget Target_7500:=[[140.174,187.004,-28.8],[1,0,0,0],[-1,0,0,1],[9E+09,9E+09,9E+09,9E+09,9E+09,9E+09]];
    CONST robtarget Target_7510:=[[141.623,187.004,-28.8],[1,0,0,0],[-1,0,0,1],[9E+09,9E+09,9E+09,9E+09,9E+09,9E+09]];
    CONST robtarget Target_7520:=[[142.676,187.003,-28.8],[1,0,0,0],[-1,0,0,1],[9E+09,9E+09,9E+09,9E+09,9E+09,9E+09]];
    CONST robtarget Target_7530:=[[143.527,187.003,-28.8],[1,0,0,0],[-1,0,0,1],[9E+09,9E+09,9E+09,9E+09,9E+09,9E+09]];

    PROC main()
        WHILE TRUE DO
            IF DI_01 = 1 THEN
                TPWrite "Iniciando protocolo de mantenimiento";
                SetDO DO_01,1;
                Mantenimiento;
                TPWrite "El robot ha llegado a posición de mantenimiento";
                SetDO DO_01,0;
            ELSEIF DI_02 = 1 THEN
                TPWrite "Iniciando protocolo de dibujo";
                SetDO DO_02,1;
                Home;
                TPWrite "Dibujando";
                Path_10;
                Path_20;
                Path_30;
                Path_40;
                Path_50;
                Path_60;
                Path_70;
                Path_80;
                Path_90;
                Path_100;
                Path_110;
                TPWrite "El robot ha acabdo de dibujar";
                TPWrite "Yendo a posición de HOME";
                Home;
                SetDO DO_02,0;
            ENDIF
        ENDWHILE
    ENDPROC

    PROC Mantenimiento()
        MoveJ Target_0,v100,fine,TCP_Marcador\WObj:=Workobject_3;
    ENDPROC

    PROC Home()
        MoveJ Target_1,v100,fine,TCP_Marcador\WObj:=Workobject_3;
    ENDPROC

    PROC Path_10()
        MoveJ Target_180,v100,fine,TCP_Marcador\WObj:=Workobject_3;
        MoveL Target_50,v100,fine,TCP_Marcador\WObj:=Workobject_3;
        MoveL Target_60,v100,fine,TCP_Marcador\WObj:=Workobject_3;
        MoveL Target_70,v100,fine,TCP_Marcador\WObj:=Workobject_3;
        MoveL Target_80,v100,fine,TCP_Marcador\WObj:=Workobject_3;
        MoveL Target_90,v100,fine,TCP_Marcador\WObj:=Workobject_3;
        MoveL Target_100,v100,fine,TCP_Marcador\WObj:=Workobject_3;
        MoveL Target_110,v100,fine,TCP_Marcador\WObj:=Workobject_3;
        MoveL Target_120,v100,fine,TCP_Marcador\WObj:=Workobject_3;
        MoveL Target_130,v100,fine,TCP_Marcador\WObj:=Workobject_3;
        MoveL Target_140,v100,fine,TCP_Marcador\WObj:=Workobject_3;
        MoveL Target_150,v100,fine,TCP_Marcador\WObj:=Workobject_3;
        MoveL Target_160,v100,fine,TCP_Marcador\WObj:=Workobject_3;
        MoveL Target_170,v100,fine,TCP_Marcador\WObj:=Workobject_3;
        MoveL Target_50,v100,fine,TCP_Marcador\WObj:=Workobject_3;
        MoveL Target_180,v100,fine,TCP_Marcador\WObj:=Workobject_3;
    ENDPROC

    PROC Path_20()
        MoveL Target_970,v100,fine,TCP_Marcador\WObj:=Workobject_3;
        MoveL Target_210,v100,fine,TCP_Marcador\WObj:=Workobject_3;
        MoveL Target_220,v100,fine,TCP_Marcador\WObj:=Workobject_3;
        MoveL Target_230,v100,fine,TCP_Marcador\WObj:=Workobject_3;
        MoveL Target_240,v100,fine,TCP_Marcador\WObj:=Workobject_3;
        MoveL Target_250,v100,fine,TCP_Marcador\WObj:=Workobject_3;
        MoveL Target_260,v100,fine,TCP_Marcador\WObj:=Workobject_3;
        MoveL Target_270,v100,fine,TCP_Marcador\WObj:=Workobject_3;
        MoveL Target_280,v100,fine,TCP_Marcador\WObj:=Workobject_3;
        MoveL Target_290,v100,fine,TCP_Marcador\WObj:=Workobject_3;
        MoveL Target_300,v100,fine,TCP_Marcador\WObj:=Workobject_3;
        MoveL Target_310,v100,fine,TCP_Marcador\WObj:=Workobject_3;
        MoveL Target_320,v100,fine,TCP_Marcador\WObj:=Workobject_3;
        MoveL Target_330,v100,fine,TCP_Marcador\WObj:=Workobject_3;
        MoveL Target_340,v100,fine,TCP_Marcador\WObj:=Workobject_3;
        MoveL Target_350,v100,fine,TCP_Marcador\WObj:=Workobject_3;
        MoveL Target_360,v100,fine,TCP_Marcador\WObj:=Workobject_3;
        MoveL Target_370,v100,fine,TCP_Marcador\WObj:=Workobject_3;
        MoveL Target_380,v100,fine,TCP_Marcador\WObj:=Workobject_3;
        MoveL Target_390,v100,fine,TCP_Marcador\WObj:=Workobject_3;
        MoveL Target_400,v100,fine,TCP_Marcador\WObj:=Workobject_3;
        MoveL Target_410,v100,fine,TCP_Marcador\WObj:=Workobject_3;
        MoveL Target_420,v100,fine,TCP_Marcador\WObj:=Workobject_3;
        MoveL Target_430,v100,fine,TCP_Marcador\WObj:=Workobject_3;
        MoveL Target_440,v100,fine,TCP_Marcador\WObj:=Workobject_3;
        MoveL Target_450,v100,fine,TCP_Marcador\WObj:=Workobject_3;
        MoveL Target_460,v100,fine,TCP_Marcador\WObj:=Workobject_3;
        MoveL Target_470,v100,fine,TCP_Marcador\WObj:=Workobject_3;
        MoveL Target_480,v100,fine,TCP_Marcador\WObj:=Workobject_3;
        MoveL Target_490,v100,fine,TCP_Marcador\WObj:=Workobject_3;
        MoveL Target_500,v100,fine,TCP_Marcador\WObj:=Workobject_3;
        MoveL Target_510,v100,fine,TCP_Marcador\WObj:=Workobject_3;
        MoveL Target_520,v100,fine,TCP_Marcador\WObj:=Workobject_3;
        MoveL Target_530,v100,fine,TCP_Marcador\WObj:=Workobject_3;
        MoveL Target_540,v100,fine,TCP_Marcador\WObj:=Workobject_3;
        MoveL Target_550,v100,fine,TCP_Marcador\WObj:=Workobject_3;
        MoveL Target_560,v100,fine,TCP_Marcador\WObj:=Workobject_3;
        MoveL Target_570,v100,fine,TCP_Marcador\WObj:=Workobject_3;
        MoveL Target_580,v100,fine,TCP_Marcador\WObj:=Workobject_3;
        MoveL Target_590,v100,fine,TCP_Marcador\WObj:=Workobject_3;
        MoveL Target_600,v100,fine,TCP_Marcador\WObj:=Workobject_3;
        MoveL Target_610,v100,fine,TCP_Marcador\WObj:=Workobject_3;
        MoveL Target_620,v100,fine,TCP_Marcador\WObj:=Workobject_3;
        MoveL Target_630,v100,fine,TCP_Marcador\WObj:=Workobject_3;
        MoveL Target_640,v100,fine,TCP_Marcador\WObj:=Workobject_3;
        MoveL Target_650,v100,fine,TCP_Marcador\WObj:=Workobject_3;
        MoveL Target_660,v100,fine,TCP_Marcador\WObj:=Workobject_3;
        MoveL Target_670,v100,fine,TCP_Marcador\WObj:=Workobject_3;
        MoveL Target_680,v100,fine,TCP_Marcador\WObj:=Workobject_3;
        MoveL Target_690,v100,fine,TCP_Marcador\WObj:=Workobject_3;
        MoveL Target_700,v100,fine,TCP_Marcador\WObj:=Workobject_3;
        MoveL Target_710,v100,fine,TCP_Marcador\WObj:=Workobject_3;
        MoveL Target_720,v100,fine,TCP_Marcador\WObj:=Workobject_3;
        MoveL Target_730,v100,fine,TCP_Marcador\WObj:=Workobject_3;
        MoveL Target_740,v100,fine,TCP_Marcador\WObj:=Workobject_3;
        MoveL Target_750,v100,fine,TCP_Marcador\WObj:=Workobject_3;
        MoveL Target_760,v100,fine,TCP_Marcador\WObj:=Workobject_3;
        MoveL Target_770,v100,fine,TCP_Marcador\WObj:=Workobject_3;
        MoveL Target_780,v100,fine,TCP_Marcador\WObj:=Workobject_3;
        MoveL Target_790,v100,fine,TCP_Marcador\WObj:=Workobject_3;
        MoveL Target_800,v100,fine,TCP_Marcador\WObj:=Workobject_3;
        MoveL Target_810,v100,fine,TCP_Marcador\WObj:=Workobject_3;
        MoveL Target_820,v100,fine,TCP_Marcador\WObj:=Workobject_3;
        MoveL Target_830,v100,fine,TCP_Marcador\WObj:=Workobject_3;
        MoveL Target_840,v100,fine,TCP_Marcador\WObj:=Workobject_3;
        MoveL Target_850,v100,fine,TCP_Marcador\WObj:=Workobject_3;
        MoveL Target_860,v100,fine,TCP_Marcador\WObj:=Workobject_3;
        MoveL Target_870,v100,fine,TCP_Marcador\WObj:=Workobject_3;
        MoveL Target_880,v100,fine,TCP_Marcador\WObj:=Workobject_3;
        MoveL Target_890,v100,fine,TCP_Marcador\WObj:=Workobject_3;
        MoveL Target_900,v100,fine,TCP_Marcador\WObj:=Workobject_3;
        MoveL Target_910,v100,fine,TCP_Marcador\WObj:=Workobject_3;
        MoveL Target_920,v100,fine,TCP_Marcador\WObj:=Workobject_3;
        MoveL Target_930,v100,fine,TCP_Marcador\WObj:=Workobject_3;
        MoveL Target_940,v100,fine,TCP_Marcador\WObj:=Workobject_3;
        MoveL Target_950,v100,fine,TCP_Marcador\WObj:=Workobject_3;
        MoveL Target_960,v100,fine,TCP_Marcador\WObj:=Workobject_3;
        MoveL Target_970,v100,fine,TCP_Marcador\WObj:=Workobject_3;
        MoveL Target_1360,v100,fine,TCP_Marcador\WObj:=Workobject_3;
        MoveL Target_1370,v100,fine,TCP_Marcador\WObj:=Workobject_3;
        MoveL Target_1380,v100,fine,TCP_Marcador\WObj:=Workobject_3;
        MoveL Target_1390,v100,fine,TCP_Marcador\WObj:=Workobject_3;
        MoveL Target_1400,v100,fine,TCP_Marcador\WObj:=Workobject_3;
        MoveL Target_1410,v100,fine,TCP_Marcador\WObj:=Workobject_3;
        MoveL Target_1420,v100,fine,TCP_Marcador\WObj:=Workobject_3;
        MoveL Target_1430,v100,fine,TCP_Marcador\WObj:=Workobject_3;
        MoveL Target_1440,v100,fine,TCP_Marcador\WObj:=Workobject_3;
        MoveL Target_1450,v100,fine,TCP_Marcador\WObj:=Workobject_3;
        MoveL Target_1460,v100,fine,TCP_Marcador\WObj:=Workobject_3;
        MoveL Target_1470,v100,fine,TCP_Marcador\WObj:=Workobject_3;
        MoveL Target_1480,v100,fine,TCP_Marcador\WObj:=Workobject_3;
        MoveL Target_1490,v100,fine,TCP_Marcador\WObj:=Workobject_3;
        MoveL Target_1500,v100,fine,TCP_Marcador\WObj:=Workobject_3;
        MoveL Target_1510,v100,fine,TCP_Marcador\WObj:=Workobject_3;
        MoveL Target_1520,v100,fine,TCP_Marcador\WObj:=Workobject_3;
        MoveL Target_1530,v100,fine,TCP_Marcador\WObj:=Workobject_3;
        MoveL Target_1580,v100,fine,TCP_Marcador\WObj:=Workobject_3;
        MoveL Target_1590,v100,fine,TCP_Marcador\WObj:=Workobject_3;
        MoveL Target_1600,v100,fine,TCP_Marcador\WObj:=Workobject_3;
        MoveL Target_1370,v100,fine,TCP_Marcador\WObj:=Workobject_3;
        MoveL Target_1360,v100,fine,TCP_Marcador\WObj:=Workobject_3;
    ENDPROC

    PROC Path_30()
        MoveL Target_1610,v100,fine,TCP_Marcador\WObj:=Workobject_3;
        MoveL Target_1620,v100,fine,TCP_Marcador\WObj:=Workobject_3;
        MoveL Target_1630,v100,fine,TCP_Marcador\WObj:=Workobject_3;
        MoveL Target_1640,v100,fine,TCP_Marcador\WObj:=Workobject_3;
        MoveL Target_1650,v100,fine,TCP_Marcador\WObj:=Workobject_3;
        MoveL Target_1660,v100,fine,TCP_Marcador\WObj:=Workobject_3;
        MoveL Target_1670,v100,fine,TCP_Marcador\WObj:=Workobject_3;
        MoveL Target_1680,v100,fine,TCP_Marcador\WObj:=Workobject_3;
        MoveL Target_1690,v100,fine,TCP_Marcador\WObj:=Workobject_3;
        MoveL Target_1700,v100,fine,TCP_Marcador\WObj:=Workobject_3;
        MoveL Target_1710,v100,fine,TCP_Marcador\WObj:=Workobject_3;
        MoveL Target_1620,v100,fine,TCP_Marcador\WObj:=Workobject_3;
        MoveL Target_1610,v100,fine,TCP_Marcador\WObj:=Workobject_3;
    ENDPROC

    PROC Path_40()
        MoveL Target_1720,v100,fine,TCP_Marcador\WObj:=Workobject_3;
        MoveL Target_1730,v100,fine,TCP_Marcador\WObj:=Workobject_3;
        MoveL Target_1740,v100,fine,TCP_Marcador\WObj:=Workobject_3;
        MoveL Target_1750,v100,fine,TCP_Marcador\WObj:=Workobject_3;
        MoveL Target_1760,v100,fine,TCP_Marcador\WObj:=Workobject_3;
        MoveL Target_1770,v100,fine,TCP_Marcador\WObj:=Workobject_3;
        MoveL Target_1780,v100,fine,TCP_Marcador\WObj:=Workobject_3;
        MoveL Target_1790,v100,fine,TCP_Marcador\WObj:=Workobject_3;
        MoveL Target_1800,v100,fine,TCP_Marcador\WObj:=Workobject_3;
        MoveL Target_1810,v100,fine,TCP_Marcador\WObj:=Workobject_3;
        MoveL Target_1820,v100,fine,TCP_Marcador\WObj:=Workobject_3;
        MoveL Target_1830,v100,fine,TCP_Marcador\WObj:=Workobject_3;
        MoveL Target_1840,v100,fine,TCP_Marcador\WObj:=Workobject_3;
        MoveL Target_1850,v100,fine,TCP_Marcador\WObj:=Workobject_3;
        MoveL Target_1860,v100,fine,TCP_Marcador\WObj:=Workobject_3;
        MoveL Target_1870,v100,fine,TCP_Marcador\WObj:=Workobject_3;
        MoveL Target_1880,v100,fine,TCP_Marcador\WObj:=Workobject_3;
        MoveL Target_1890,v100,fine,TCP_Marcador\WObj:=Workobject_3;
        MoveL Target_1900,v100,fine,TCP_Marcador\WObj:=Workobject_3;
        MoveL Target_1910,v100,fine,TCP_Marcador\WObj:=Workobject_3;
        MoveL Target_1920,v100,fine,TCP_Marcador\WObj:=Workobject_3;
        MoveL Target_1930,v100,fine,TCP_Marcador\WObj:=Workobject_3;
        MoveL Target_1940,v100,fine,TCP_Marcador\WObj:=Workobject_3;
        MoveL Target_1950,v100,fine,TCP_Marcador\WObj:=Workobject_3;
        MoveL Target_1960,v100,fine,TCP_Marcador\WObj:=Workobject_3;
        MoveL Target_1970,v100,fine,TCP_Marcador\WObj:=Workobject_3;
        MoveL Target_1980,v100,fine,TCP_Marcador\WObj:=Workobject_3;
        MoveL Target_1990,v100,fine,TCP_Marcador\WObj:=Workobject_3;
        MoveL Target_2000,v100,fine,TCP_Marcador\WObj:=Workobject_3;
        MoveL Target_2010,v100,fine,TCP_Marcador\WObj:=Workobject_3;
        MoveL Target_2020,v100,fine,TCP_Marcador\WObj:=Workobject_3;
        MoveL Target_2030,v100,fine,TCP_Marcador\WObj:=Workobject_3;
        MoveL Target_2040,v100,fine,TCP_Marcador\WObj:=Workobject_3;
        MoveL Target_2050,v100,fine,TCP_Marcador\WObj:=Workobject_3;
        MoveL Target_1730,v100,fine,TCP_Marcador\WObj:=Workobject_3;
        MoveL Target_1720,v100,fine,TCP_Marcador\WObj:=Workobject_3;
    ENDPROC

    PROC Path_50()
        MoveL Target_2060,v100,fine,TCP_Marcador\WObj:=Workobject_3;
        MoveL Target_2070,v100,fine,TCP_Marcador\WObj:=Workobject_3;
        MoveL Target_2080,v100,fine,TCP_Marcador\WObj:=Workobject_3;
        MoveL Target_2090,v100,fine,TCP_Marcador\WObj:=Workobject_3;
        MoveL Target_2100,v100,fine,TCP_Marcador\WObj:=Workobject_3;
        MoveL Target_2110,v100,fine,TCP_Marcador\WObj:=Workobject_3;
        MoveL Target_2120,v100,fine,TCP_Marcador\WObj:=Workobject_3;
        MoveL Target_2130,v100,fine,TCP_Marcador\WObj:=Workobject_3;
        MoveL Target_2140,v100,fine,TCP_Marcador\WObj:=Workobject_3;
        MoveL Target_2150,v100,fine,TCP_Marcador\WObj:=Workobject_3;
        MoveL Target_2160,v100,fine,TCP_Marcador\WObj:=Workobject_3;
        MoveL Target_2170,v100,fine,TCP_Marcador\WObj:=Workobject_3;
        MoveL Target_2180,v100,fine,TCP_Marcador\WObj:=Workobject_3;
        MoveL Target_2190,v100,fine,TCP_Marcador\WObj:=Workobject_3;
        MoveL Target_2200,v100,fine,TCP_Marcador\WObj:=Workobject_3;
        MoveL Target_2210,v100,fine,TCP_Marcador\WObj:=Workobject_3;
        MoveL Target_2220,v100,fine,TCP_Marcador\WObj:=Workobject_3;
        MoveL Target_2230,v100,fine,TCP_Marcador\WObj:=Workobject_3;
        MoveL Target_2240,v100,fine,TCP_Marcador\WObj:=Workobject_3;
        MoveL Target_2250,v100,fine,TCP_Marcador\WObj:=Workobject_3;
        MoveL Target_2070,v100,fine,TCP_Marcador\WObj:=Workobject_3;
        MoveL Target_2060,v100,fine,TCP_Marcador\WObj:=Workobject_3;
        MoveL Target_2260,v100,fine,TCP_Marcador\WObj:=Workobject_3;
        MoveL Target_2270,v100,fine,TCP_Marcador\WObj:=Workobject_3;
        MoveL Target_2280,v100,fine,TCP_Marcador\WObj:=Workobject_3;
        MoveL Target_2290,v100,fine,TCP_Marcador\WObj:=Workobject_3;
        MoveL Target_2300,v100,fine,TCP_Marcador\WObj:=Workobject_3;
        MoveL Target_2310,v100,fine,TCP_Marcador\WObj:=Workobject_3;
        MoveL Target_2320,v100,fine,TCP_Marcador\WObj:=Workobject_3;
        MoveL Target_2330,v100,fine,TCP_Marcador\WObj:=Workobject_3;
        MoveL Target_2340,v100,fine,TCP_Marcador\WObj:=Workobject_3;
        MoveL Target_2350,v100,fine,TCP_Marcador\WObj:=Workobject_3;
        MoveL Target_2360,v100,fine,TCP_Marcador\WObj:=Workobject_3;
        MoveL Target_2370,v100,fine,TCP_Marcador\WObj:=Workobject_3;
        MoveL Target_2270,v100,fine,TCP_Marcador\WObj:=Workobject_3;
        MoveL Target_2260,v100,fine,TCP_Marcador\WObj:=Workobject_3;
    ENDPROC

